// TwinCAT 3 PLC project L2SIVacuum
// Title: LCLS Vacuum
// Company: SLAC - LCLS
// Author: LCLS ECS-Platforms
// ProjectVersion: 0.0.0.0.0.0.
// ProgramVersion: 3.1.4026.17
// libraries:
//   LCLS General, * (SLAC)
//   PMPS, * (SLAC - LCLS)
//   Tc2_DataExchange, * (Beckhoff Automation GmbH)
//   Tc2_EtherCAT, * (Beckhoff Automation GmbH)
//   Tc2_ModbusSrv, * (Beckhoff Automation GmbH)
//   Tc2_SerialCom, * (Beckhoff Automation GmbH)
//   Tc2_Standard, * (Beckhoff Automation GmbH)
//   Tc2_System, * (Beckhoff Automation GmbH)
//   Tc2_TcpIp, * (Beckhoff Automation GmbH)
//   Tc2_Utilities, * (Beckhoff Automation GmbH)
//   Tc3_EventLogger, * (Beckhoff Automation GmbH)
//   Tc3_JsonXml, * (Beckhoff Automation GmbH)
//   Tc3_Module, * (Beckhoff Automation GmbH)
//   TcUnit, * (www.tcunit.org)
// project tree:
//   DUTs/Gauges/ E_PressureState.TcDUT (not stored), Gauge_Type.TcDUT (not stored), ST_VG.TcDUT (not stored)
//   DUTs/LVDT/ ST_SerLVC4000.TcDUT (not stored)
//   DUTs/Oerlikon/ ST_TD20Status.TcDUT (not stored), ST_TD400Control.TcDUT (not stored), ST_TD400Status.TcDUT (not stored)
//   DUTs/Pfeiffer/ ST_PfeifferControl.TcDUT (not stored), ST_PfeifferStatus.TcDUT (not stored)
//   DUTs/Pumps/ E_PumpState.TcDUT (not stored), ST_AgilentPTM.TcDUT (not stored), ST_EbaraDryPump.TcDUT (not stored), ST_EbaraEVA.TcDUT, ST_EbaraPTM.TcDUT (not stored), ST_KashiyamaDryPump.TcDUT (not stored), ST_LeyboldPTM.TcDUT (not stored), ST_PfeifferPTM.TcDUT (not stored), ST_PIP.TcDUT (not stored), ST_PTM.TcDUT (not stored), ST_RoughPump.TcDUT (not stored)
//   DUTs/Valves/ E_ValvePositionState.TcDUT (not stored), E_VCN.TcDUT (not stored), E_2OO3_MODE.TcDUT (not stored), E_VGC.TcDUT (not stored), ST_ValveBase.TcDUT (not stored), ST_VFS.TcDUT (not stored), ST_VGC_2S.TcDUT (not stored), ST_VRC_NO.TcDUT (not stored), ST_VWC_NO.TcDUT (not stored), ST_VVC.TcDUT (not stored), ST_VCC_NO.TcDUT (not stored), ST_VCN.TcDUT (not stored), ST_VGC.TcDUT (not stored), ST_VRC.TcDUT (not stored)
//   DUTs/Valves/VAT590/EtherCAT Interface/ E_ControlMode.TcDUT (not stored), E_ControlModeSP.TcDUT (not stored), E_FatalErrors.TcDUT (not stored), ST_ExtendedWarnings.TcDUT (not stored), ST_GeneralControlSP.TcDUT (not stored), ST_GeneralStatus.TcDUT (not stored), ST_GeneralWarnings.TcDUT (not stored)
//   DUTs/Valves/VAT590/ E_VAT590_AccessMode.TcDUT (not stored), E_VAT590_PID_CTRL.TcDUT (not stored), E_VCN_VAT590.TcDUT (not stored), ST_CoEIndSub.TcDUT (not stored), ST_VAT590_COE.TcDUT, ST_VAT590_STATUS.TcDUT (not stored), ST_VCN_VAT590.TcDUT
//   GVLs/ Constants.TcGVL (not stored), Global_Variables.TcGVL (not stored), GVL_MacroSensorsParameters.TcGVL (not stored), GVL_PfeifferParameters.TcGVL (not stored)
//   / PlcTask.TcTTO (not stored)
//   POUs/ADS/ FB_ADS.TcPOU (not stored), FB_ADS_WATCHDOG.TcPOU (not stored), FB_TBOOL_ADS.TcPOU (not stored)
//   POUs/Functions/Deprecated/Gauges/ FB_MKS317A.TcPOU (not stored), FB_MKS500_EP.TcPOU (not stored), FB_PressureState.TcPOU (not stored)
//   POUs/Functions/Deprecated/Valves/ FB_VCC.TcPOU (not stored), FB_VCC_NO.TcPOU (not stored), FB_VGC_AP.TcPOU (not stored), FB_VGC_EBD.TcPOU (not stored)
//   POUs/Functions/Gauges/ FB_901_ECAT.TcPOU (not stored), FB_9XX.TcPOU (not stored), FB_972.TcPOU (not stored), FB_IE514.TcPOU (not stored), FB_MX7M.TcPOU (not stored), FB_MKS355.TcPOU (not stored), FB_GaugeBase.TcPOU (not stored), FB_CVM201.TcPOU (not stored), FB_CCM501.TcPOU (not stored), FB_IMG401.TcPOU (not stored), FB_MKS909.TcPOU (not stored), FB_MKS909_RBK.TcPOU (not stored), FB_CMR362.TcPOU (not stored), FB_GCM.TcPOU (not stored), FB_ITR90.TcPOU (not stored), FB_MKS392.TcPOU (not stored), FB_MKS500.TcPOU (not stored), FB_MKS722.TcPOU (not stored), FB_MKS_937A.TcPOU (not stored), FB_MKS317.TcPOU (not stored), FB_MKS275.TcPOU (not stored), FB_MKS_937B.TcPOU (not stored), FB_MKS422.TcPOU (not stored)
//   POUs/Functions/Gauges/Interfaces/ FB_GaugeModbus.TcPOU (not stored), FB_Gauge_Interface.TcPOU (not stored), FB_TGCC_ADS.TcPOU (not stored), FB_TGPI_ADS.TcPOU (not stored), FB_GaugeSelection.TcPOU (not stored)
//   POUs/Functions/Pumps/ FB_EbaraDryPump.TcPOU (not stored), FB_EbaraEVA.TcPOU, FB_KashiyamaPump.TcPOU (not stored), FB_KashiyamaPump_G.TcPOU (not stored), FB_PIP_Gamma.TcPOU (not stored), FB_PIP_Gamma_V2.TcPOU, FB_PIP_SIP.TcPOU (not stored), FB_PTM_Agilent.TcPOU (not stored), FB_PTM_Ebara_011M.TcPOU (not stored), FB_PTM_Ebara_010M.TcPOU (not stored), FB_PTM_MagDriveDigital.TcPOU (not stored), FB_PTM_Pfeiffer.TcPOU, FB_PTM_TurboDrive.TcPOU, FB_PTM_TwisTorr.TcPOU (not stored), FB_Pump.TcPOU (not stored), FB_ScrollPump.TcPOU (not stored)
//   POUs/Functions/Pumps/functions/ FB_TurboExtLogic.TcPOU (not stored), F_TurboExtILK_NO.TcPOU (not stored), F_TurboExtILKLogic.TcPOU (not stored), F_TurboExtILKLogic_2.TcPOU (not stored), F_TurboExtILK_NO_1.TcPOU (not stored)
//   POUs/Functions/Pumps/Interfaces/ FB_PIP_Interface_In.TcPOU (not stored), FB_PIP_Interface_Out.TcPOU (not stored), FB_TPIP_ADS.TcPOU (not stored)
//   POUs/Functions/Valves/ FB_Kashiyama_VRC.TcPOU (not stored), FB_MKS248.TcPOU (not stored), FB_TurbVentvalve_NO.TcPOU (not stored), FB_Valve.TcPOU (not stored), FB_VCN_VAT590.TcPOU, FB_VFS.TcPOU (not stored), FB_VFS_2OO3.TcPOU, FB_VGC_NEW.TcPOU, FB_VGC_2S.TcPOU (not stored), FB_VRC_DA.TcPOU (not stored), FB_VRC_EBD.TcPOU (not stored), FB_VRC_NC_ClsLS.TcPOU (not stored), FB_VRC_NO.TcPOU (not stored), FB_VRC_NO_FFO.TcPOU (not stored), FB_VVC.TcPOU (not stored), FB_VCN.TcPOU (not stored), FB_VGC.TcPOU (not stored), FB_VRC.TcPOU (not stored), FB_VRC_OK_CLS.TcPOU (not stored)
//   POUs/Functions/Valves/functions/ F_RoughPumpInlet_ILK.TcPOU (not stored), F_TurboGateValve_ILK.TcPOU (not stored), F_TurboGateValve_ILK_1.TcPOU (not stored), F_TurboGateValve_Protection_ILK.TcPOU (not stored), F_TURBO_VRC_ILK.TcPOU (not stored), F_VALVE_REL_ILK.TcPOU (not stored), F_VRC_DIODE_ILK_OK.TcPOU (not stored), F_VRC_DIODE_ILK.TcPOU (not stored)
//   POUs/Functions/Valves/Interfaces/ FB_TVGC_2S_ADS.TcPOU (not stored), FB_VFS_2OO3Interface.TcPOU, FB_VFS_Interface.TcPOU, FB_TVGC_ADS.TcPOU (not stored), FB_Valve_Interface.TcPOU (not stored), ITF_Valve.TcIO (not stored)
//   POUs/Serial drivers/LVDT/MacroSensors/ FB_LVC4000Com.TcPOU (not stored), FB_LVC4000SerialDriver.TcPOU (not stored), FB_LVC4000Transaction.TcPOU (not stored)
//   POUs/Serial drivers/Pumps/Oerlikon TD20/ FB_OERLIKON_TD20_COM.TcPOU (not stored), FB_OERLIKON_TO_PTM.TcPOU (not stored), FB_TD20SerialDriver.TcPOU (not stored), FB_TD20Transaction.TcPOU (not stored), F_CalcTD20Checksum.TcPOU (not stored)
//   POUs/Serial drivers/Pumps/Oerlikon TD400/ FB_OERLIKON_TD400_COM.TcPOU (not stored), FB_OERLIKON_TD400_TO_PTM.TcPOU (not stored), FB_TD400SerialDriver.TcPOU (not stored), FB_TD400Transaction.TcPOU (not stored), F_CalcTD400Checksum.TcPOU (not stored)
//   POUs/Serial drivers/Pumps/Pfeiffer/ FB_PfeifferSerialDriver.TcPOU (not stored), FB_PfeifferTransaction.TcPOU (not stored), FB_PFEIFFER_COM.TcPOU (not stored), FB_PFEIFFER_TO_PTM.TcPOU (not stored), F_CalcPfeifferCheckSum.TcPOU (not stored)
//   UnitTests/Functions/ V_TO_INT.TcPOU (not stored)
//   UnitTests/Gauges/ FB_GCC_Test.TcPOU (not stored), FB_GHC_Test.TcPOU (not stored), FB_GPI_Test.TcPOU (not stored)
//   UnitTests/ PRG_Test.TcPOU (not stored)
//   UnitTests/Pumps/ FB_PIP_Test.TcPOU (not stored), FB_PTM_Test.TcPOU (not stored)
//   UnitTests/Valves/ FB_VGC_Test.TcPOU (not stored), FB_VRC_Test.TcPOU (not stored)
//   Version/ Global_Version.TcGVL
// real-time tasks:
//   TASK TestTask: cycle T#10ms, priority 16, ADS port 350
// variable links:
//   L2SIVacuum/L2SIVacuum Instance <-> L2SIVacuum/L2SIVacuum Instance
//     PlcTask Inputs/PRG_Test.fb_GCC_Test.fb_MKS422.i_iPRESS_R <-> PlcTask Outputs/PRG_Test.fb_GCC_Test.i_iPRESS_R
//     PlcTask Inputs/PRG_Test.fb_GPI_Test.fb_MKS275.i_iPRESS_R <-> PlcTask Outputs/PRG_Test.fb_GPI_Test.i_iPRESS_R
//     PlcTask Inputs/PRG_Test.fb_GPI_Test.fb_MKS317.i_iPRESS_R <-> PlcTask Outputs/PRG_Test.fb_GPI_Test.i_iPRESS_R
//     PlcTask Inputs/PRG_Test.fb_PTM_Test.fb_PTM_Ebara_010M.i_iCurrentMon <-> PlcTask Outputs/PRG_Test.fb_PTM_Test.i_iCurrentMon
//     PlcTask Inputs/PRG_Test.fb_PTM_Test.fb_PTM_Ebara_010M.i_iRawSpeed <-> PlcTask Outputs/PRG_Test.fb_PTM_Test.i_iRawSpeed
//     PlcTask Inputs/PRG_Test.fb_PTM_Test.fb_PTM_Ebara_010M.i_iTempMon <-> PlcTask Outputs/PRG_Test.fb_PTM_Test.i_iTempMon
//     PlcTask Inputs/PRG_Test.fb_PTM_Test.q_iSpeedSet <-> PlcTask Outputs/PRG_Test.fb_PTM_Test.i_diCurSpd

// ---- DUTs/Pumps/ST_EbaraEVA.TcDUT
TYPE ST_EbaraEVA EXTENDS ST_RoughPump:
STRUCT

(* Output *)
    //q_xRunDO 	:	BOOL; in Rough PUMP


(* Input *)
{attribute 'pytmc' := '
    pv: REMOTE;
    field: ZNAM FALSE;
    field: ONAM TRUE;
    io: io;
    '}
    q_xRemote	:	BOOL;
    {attribute 'pytmc' := '
    pv: ALARM_OK;
    field: ZNAM FALSE;
    field: ONAM TRUE;
    io: i
    '}
    i_xAlarmOK	:	BOOL;

    {attribute 'pytmc' := '
    pv: RUN_DI;
    field: ZNAM FALSE;
    field: ONAM TRUE;
    io: i
    '}
    i_xIsRun		:	BOOL;



END_STRUCT
END_TYPE

// ---- DUTs/Valves/VAT590/ST_VAT590_COE.TcDUT
TYPE ST_VAT590_COE :
STRUCT
    {attribute 'pytmc' := '
    pv: PID_CTRL
    io: io
    '}
    ePIDCtrl: E_VAT590_PID_CTRL;
    (*Adaptive Downstream Parameters*)
    {attribute 'pytmc' := '
    pv: SENS_DELAY_AD
    io: io
    field: EGU "s"
    field: DRVL 0.0
    field: DRVH 1.0
    '}
    fSensorDelay_AD : REAL;
    {attribute 'pytmc' := '
    pv: RAMP_TIME_AD
    io: io
    field: EGU "s"
    field: DRVL 0.0
    field: DRVH 1000000.0
    '}
    fRampTime_AD : REAL;
    {attribute 'pytmc' := '
    pv: RAMP_MODE_AD
    io: io
    field: ZNAM CONST_TIME
    field: ONAM CONST_SLOPE
    '}
    bRampMode_AD : BOOL;
    {attribute 'pytmc' := '
    pv: GAIN_FACTOR_AD
    io: io
    field: PREC 4
    field: DRVL 0.0001
    field: DRVH 7.5
    '}
    fGainFactor_AD : REAL;
    (*Fixed 1 Parameters*)
    {attribute 'pytmc' := '
    pv: RAMP_TIME_FIX1
    io: io
    field: EGU "s"
    field: DRVL 0.0
    field: DRVH 1000000.0
    '}
    fRampTime_FIX1 : REAL;
    {attribute 'pytmc' := '
    pv: RAMP_MODE_FIX1
    io: io
    field: ZNAM CONST_TIME
    field: ONAM CONST_SLOPE
    '}
    bRampMode_FIX1 : BOOL;
    {attribute 'pytmc' := '
    pv: CTRL_DIR_FIX1
    io: io
    field: ZNAM DOWNSTREAM
    field: ONAM UPSTREAM
    '}
    bCtrlDir_FIX1 : BOOL;
    {attribute 'pytmc' := '
    pv: PGAIN_FIX1
    io: io
    field: DRVL 0.001
    field: DRVH 100.0
    '}
    fPGain_FIX1 : REAL;
    {attribute 'pytmc' := '
    pv: IGAIN_FIX1
    io: io
    field: DRVL 0.0
    field: DRVH 100.0
    '}
    fIGain_FIX1 : REAL;
    (*Fixed 2 Parameters*)
    {attribute 'pytmc' := '
    pv: RAMP_TIME_FIX2
    io: io
    field: EGU "s"
    field: DRVL 0.0
    field: DRVH 1000000.0
    '}
    fRampTime_FIX2 : REAL;
    {attribute 'pytmc' := '
    pv: RAMP_MODE_FIX2
    io: io
    field: ZNAM CONST_TIME
    field: ONAM CONST_SLOPE
    '}
    bRampMode_FIX2 : BOOL;
    {attribute 'pytmc' := '
    pv: CTRL_DIR_FIX2
    io: io
    field: ZNAM DOWNSTREAM
    field: ONAM UPSTREAM
    '}
    bCtrlDir_FIX2 : BOOL;
    {attribute 'pytmc' := '
    pv: PGAIN_FIX2
    io: io
    field: DRVL 0.001
    field: DRVH 100.0
    '}
    fPGain_FIX2 : REAL;
    {attribute 'pytmc' := '
    pv: IGAIN_FIX2
    io: io
    field: DRVL 0.0
    field: DRVH 100.0
    '}
    fIGain_FIX2 : REAL;
    (*Soft Pump Parameters*)
    {attribute 'pytmc' := '
    pv: RAMP_TIME_SP
    io: io
    field: EGU "s"
    field: DRVL 0.0
    field: DRVH 1000000.0
    '}
    fRampTime_SP : REAL;
    {attribute 'pytmc' := '
    pv: RAMP_MODE_SP
    io: io
    field: ZNAM CONST_TIME
    field: ONAM CONST_SLOPE
    '}
    bRampMode_SP : BOOL;
    {attribute 'pytmc' := '
    pv: PGAIN_SP
    io: io
    field: DRVL 0.001
    field: DRVH 100.0
    '}
    fPGain_SP : REAL;
END_STRUCT
END_TYPE

// ---- DUTs/Valves/VAT590/ST_VCN_VAT590.TcDUT
TYPE ST_VCN_VAT590 :
STRUCT
    (* VCN - Valve Controlled Needle
    Used for VAT590 needle valves *)
    {attribute 'pytmc' := '
    pv: POS_RAW
    io: i
    '}
    nRawPosition : DINT; //Position readback
    {attribute 'pytmc' := '
    pv: PRES_RAW
    io: i
    '}
    nRawPressure : DINT; //Pressure readback
    {attribute 'pytmc' := '
    pv: PRES_TORR
    field: EGU "TORR"
    io: i
    '}
    fPressure : REAL; //Pressure readback in Torr units
    {attribute 'pytmc' := '
    pv: POS_SP
    io: i
    '}
    nPositionSP : DINT; //Position setpoint readback
    {attribute 'pytmc' := '
    pv: PRES_SP
    io: i
    '}
    nPressureSP : DINT; //Pressure setpoint readback
    {attribute 'pytmc' := '
    pv: ILK_OK
    field: ZNAM NOT OK
    field: ONAM OK
    field: ZSV MAJOR
    field: OSV NO_ALARM
    io: i
    '}
    bIlkOK : BOOL := FALSE; //Interlock Bit status
    {attribute 'pytmc' := '
    pv: POS_LIMIT
    io: io
    autosave_pass1: VAL DESC
    '}
    fPosSetLimit	: REAL := 100; //Percentage Upper limit on valve open
    {attribute 'pytmc' := '
    pv: PRES_SET_LIMIT
    io: io
    autosave_pass1: VAL DESC
    '}
    fPresSetLimit	: REAL := 1E-2; //Upper limit for pressure control
    {attribute 'pytmc' := '
    pv: PRES_RDBK_LIMIT
    io: io
    autosave_pass1: VAL DESC
    '}
    fPresRdbkLimit : REAL := 1E-4;  //Upper limit for pressure reading before valve close
    {attribute 'pytmc' := '
    pv: POS_REQ
    field: DRVL 0.0
    field: DRVH 100.0
    io: io
    '}
    fReqPosition : REAL; //Requested position (0.0-100.0%)
    {attribute 'pytmc' := '
    pv: PRES_REQ
    field: EGU "TORR"
    io: io;
    '}
    fReqPressure : REAL; //Requested pressure in Torr units
    {attribute 'pytmc' :=  '
    pv: STATE
    io: io
    '}
    eValveControl : E_VCN_VAT590; //Valve control mode
    {attribute 'pytmc' := '
    pv:
    '}
    stValveStatus : ST_VAT590_STATUS; //All Valve status readbacks
    {attribute 'pytmc' :=  '
    pv: PRES_SENS
    io: io
    '}
    ePressureSensor : E_VAT590_PressureSensor; //Select pressure sensor
    {attribute 'pytmc' :=  '
    pv: REM_CTRL
    io: io
    '}
    eRemoteControl : E_VAT590_AccessMode; //Select remote control mode
    {attribute 'pytmc' := '
    pv: ZERO
    io: io
    '}
    bZero : BOOL; //Activate Zero function bit
    {attribute 'pytmc' := '
    pv: COE_PARAM
    '}
    stCoeParameters : ST_VAT590_COE; //Coe Parameters
    {attribute 'pytmc' := '
    pv: COE_ERROR
    field: ZNAM OK
    field: ONAM ERROR
    field: ZSV NO_ALARM
    field: OSV MINOR
    io: i
    '}
    bCoeError : BOOL; //Coe Interface Error
    {attribute 'pytmc' := '
    pv: COE_RESET
    io: io
    '}
    bResetCoeError : BOOL; //Reset Coe Interface Error
    {attribute 'pytmc' := '
    pv: ETHCAT_COMM_STATUS
    field: ZNAM OK
    field: ONAM ERROR
    field: ZSV NO_ALARM
    field: OSV MAJOR
    io: i
    '}
    bValveEthCatStatus : BOOL; //Status of the Ethercat Communication with device
END_STRUCT
END_TYPE

// ---- Version/Global_Version.TcGVL
{attribute 'TcGenerated'}
{attribute 'no-analysis'}
{attribute 'linkalways'}
// This function has been automatically generated from the project information.
VAR_GLOBAL CONSTANT
	{attribute 'const_non_replaced'}
	stLibVersion_LCLS_Vacuum : ST_LibVersion := (iMajor := 0, iMinor := 0, iBuild := 0, iRevision := 1, nFlags := 0, sVersion := '0.0.0.1');
END_VAR

// ---- POUs/Functions/Pumps/FB_EbaraEVA.TcPOU
(*This function block does basic controls for the Ebara EV-A  pump. Turns off pump
in the event of errors/ warnings. Provides interlocking interface.*)
FUNCTION_BLOCK FB_EbaraEVA EXTENDS FB_Pump
VAR_INPUT
    i_xExtIlkOK	:	BOOL;
END_VAR
VAR_OUTPUT
    {attribute 'pytmc' := '
    pv:
    '}
    stPump	:	ST_EbaraEVA; //Ebara dry pump structure
END_VAR
VAR
  // For logging
  (*  fbLogger : FB_LogMessage := (eSubsystem:=E_SubSystem.VACUUM);
    ePrevState : E_PumpState;
    tErrorPresent : R_TRIG;
    tAction : R_TRIG; // Primary action of this device (OPN_DO, PUMP_RUN, etc.)
    tFault : F_TRIG;*)

(*IO*)
    q_xRunDo AT%Q* : BOOL; // Output signal
    q_xRemote At%Q* :BOOL;// Remote/Local Control
    q_xResetAlarm At%Q* :BOOL;// Remote/Local Control
    i_xAlarmOK AT%I* :BOOL; // Normally closed Alarm bit
    i_xIsRun   AT%I*:BOOL; // Input status
END_VAR

(*MG 2019*)
stPump.xIlkOK := i_xExtIlkOK AND stPump.i_xAlarmOK ;
// Enable the remote signal when the interlock evaluation is ok
//stPump.q_xRemote := stPump.xIlkOK;

IF stPump.xIlkOK THEN
    stPump.q_xRunDO := stPump.pv_xRunSW;
    stPump.q_xRemote := stPump.pv_xRunSW;
ELSE
        stPump.PV_xRunSW := FALSE;
        stPump.q_xRunDO := FALSE;
END_IF

(*State evaluation*)
IF NOT(stPump.i_xAlarmOK ) THEN
     ePrevState := stpump.eState;
    stpump.eState := pumpFAULT;
ELSIF NOT stpump.q_xRunDo AND stPump.i_xAlarmOK THEN
        stpump.eState := pumpSTOPPED;
ELSIF NOT stpump.q_xRunDo AND NOT stPump.i_xIsRun THEN
        stpump.eState := pumpSTARTING;
ELSIF stPump.i_xIsRun THEN
        stpump.eState := pumpRUNNING;
ELSE
    stpump.eState := pumpFAULT;
END_IF


//Soft IO Mapping
ACT_IO();

// Log States and triggers
ACT_Logger();

ACTION ACT_IO:
stPump.i_xAlarmOK:=	i_xAlarmOK;
stPump.xErr:=	NOT(i_xAlarmOK);
stPump.i_xIsRun := i_xIsRun;
(*outputs*)
q_xRunDo:=stPump.q_xRunDo;
q_xRemote:= stPump.q_xRemote;
END_ACTION

ACTION ACT_Logger:
// ILK logger
IF NOT i_xExtIlkOK AND ePrevState = pumpRUNNING THEN
         fbLogger(sMsg:='Lost external interlock while pump was running.', eSevr:=TcEventSeverity.Critical);
END_IF

//STATE Logger
IF ePrevState <> stpump.eState THEN
      CASE stpump.eState OF
        pumpFAULT:
            fbLogger(sMsg:='Pump Fault.', eSevr:=TcEventSeverity.Critical);
          pumpSTOPPED:
            fbLogger(sMsg:='Pump stopped.', eSevr:=TcEventSeverity.Critical);
        pumpSTARTING:
            fbLogger(sMsg:='Pump starting.', eSevr:=TcEventSeverity.Info);
        pumpRUNNING:
            fbLogger(sMsg:='Pump running.', eSevr:=TcEventSeverity.Info);
      END_CASE
      ePrevState := stpump.eState;
  END_IF

// Log Action
tAction(CLK:=  stPump.q_xRunDo);
IF tAction.Q THEN fbLogger(sMsg:='Pump commanded to start', eSevr:=TcEventSeverity.Info); END_IF


// Log FAULT
tFault(CLK:= stPump.i_xAlarmOK);
IF tFault.Q THEN fbLogger(sMsg:='Pump Lost Alarm OK bit', eSevr:=TcEventSeverity.Critical); END_IF
END_ACTION

END_FUNCTION_BLOCK

// ---- POUs/Functions/Pumps/FB_PIP_Gamma_V2.TcPOU
(* This function block does basic controls FOR the ION pump connected to a Gamma QPCe controller. *)
{attribute 'reflection'}
FUNCTION_BLOCK FB_PIP_Gamma_V2 Extends FB_Pump
VAR_INPUT
END_VAR
VAR_OUTPUT
    {attribute 'pytmc' := '
    pv:
    '}
    stPump	:	ST_PIP; //Gamma Ion pump structure
    q_IG	:	ST_VG; //When ion pump is used as a measuring device for interlocking gate valves
END_VAR
VAR
    rPRESS : REAL;

    rV : REAL;

    (* IO Controls *)
    i_iPRESS  AT %I*: INT;  //
    i_xSP_DI  AT %I* : BOOL; // NO contact //function of relay set on the QPC to HV output state

    // For logging
    tPumpErrorTimeout : TON := (PT:=T#10S); // Timeout pump start if pressure < 1E-11 for more than 10s.

    {attribute 'instance-path'}
    {attribute 'noinit'}
    sPath: STRING;
    fbGetCurTaskIdx  : GETCURTASKINDEX;
    fbWritePersistentData           : WritePersistentData;

END_VAR
VAR CONSTANT
    rMaxPressure : REAL :=1E-4; // Default protection setpoint as per the gamma QPCe manual
    rMinPressure : REAL :=1E-11;
END_VAR
VAR PERSISTENT
END_VAR

(*Pump STATE*)
tPumpErrorTimeout(IN:=(q_IG.rPRESS <= rMinPressure AND stPump.i_xHV_DI));

IF q_IG.rPRESS <= rMinPressure AND stPump.i_xHV_DI THEN
    IF tPumpErrorTimeout.Q THEN
        stPump.eState := pumpFAULT;
        tPumpErrorTimeout(IN:=FALSE);
    END_IF
ELSIF q_IG.rPRESS <= rMinPressure AND NOT stPump.i_xHV_DI THEN
    stPump.eState := pumpSTOPPED;
ELSIF stPump.i_xHV_DI THEN
    stPump.eState := pumpRUNNING;
ELSE
    stPump.eState := pumpFAULT;
END_IF

(*Update output gauge values*)
ACT_SetGauge();
(*Soft IO Mapping*)
IO();
// Log States and triggers
ACT_Logger();

ACTION ACT_Logger:
//STATE Logger
IF ePrevState <> stPump.eState THEN
      CASE stPump.eState OF
        pumpFAULT:
            fbLogger(sMsg:='Pump Fault.', eSevr:=TcEventSeverity.Critical);
        pumpSTOPPED:
            fbLogger(sMsg:='Pump stopped.', eSevr:=TcEventSeverity.Critical);
        pumpRUNNING:
            fbLogger(sMsg:='Pump running.', eSevr:=TcEventSeverity.Info);
      END_CASE
      ePrevState := stPump.eState;
  END_IF
END_ACTION

ACTION ACT_SetGauge:
(*MG*)
(* convert the analog input into readable pressure*)
(* use logarithmic Pressure calculation, Output= Normal and Offset = 0*)
rV := 10*INT_TO_REAL(i_iPress)/32767;
//Manual Page 9

if (stPump.bOutputInverted) THEN
    rPRESS := LREAL_TO_REAL(EXPT(10,(rV-stPump.iOffset)*-1));
ELSE
    rPRESS := LREAL_TO_REAL(EXPT(10,(rV-stPump.iOffset)));
END_IF

q_IG.rPRESS := rPRESS;
stPump.rPRESS := rPRESS;

IF stPump.eState := pumpRUNNING THEN
    q_IG.xPRESS_OK := TRUE;
ELSE
    q_IG.xPRESS_OK := FALSE;
END_IF

q_IG.sPath := This^.stPump.sPath;
END_ACTION

ACTION IO:
stPump.xError := (stPump.eState = pumpFAULT);

(*inputs*)
stPump.i_iPRESS:=	i_iPRESS;
stPump.i_xHV_DI:=	i_xSP_DI;

 This^.stPump.sPath:= sPath;
END_ACTION

END_FUNCTION_BLOCK

// ---- POUs/Functions/Pumps/FB_PTM_Pfeiffer.TcPOU
(* This function block does basic controls FOR the Pfeiffer Turbo pump connected to the TM700 and TC400 Controllers.
 Turns off pump in the event of errors/ warnings. Provides interlocking interface.*)
FUNCTION_BLOCK FB_PTM_Pfeiffer EXTENDS FB_Pump
VAR_INPUT
    i_xExtIlkOK : BOOL; // Connect to external interlock logic, TRUE if not used.
END_VAR
VAR_OUTPUT
    {attribute 'pytmc' := '
    pv:
    '}
    iq_stPTM : ST_PfeifferPTM;
END_VAR
VAR
    TOF_RESET: TON :=(PT:=T#1S);
    (*IO*)
    i_xAtSpd AT%I*: BOOL; // Normaml operation when true
    i_xFaultNC AT%I*: BOOL; // Error
    i_xWarn AT%I*: BOOL;
     i_xRemote AT%I*: BOOL;

    q_RunDO AT%Q*: BOOL; // Start/Stop for TC110 link this output to the Pumping station bit
    q_PumpingStation AT%Q*: BOOL; // Start/Stop interlock
    q_xRemote AT%Q*: BOOL;
    q_xReset AT%Q*: BOOL;
END_VAR

(* Basic pump supervisory section *)

q_xRemote := TRUE;
(* Interlock Sum *)
iq_stPtm.xExtRunOk:= i_xExtILKOk;
//For compatability with TC110
(*IF iq_stPTM.xExtRunOk THEN
    q_PumpingStation:= TRUE;
ELSE
    q_PumpingStation:= FALSE;
END_IF*)

IF iq_stPTM.xExtRunOk AND NOT (iq_stPTM.i_xFault) (*OR iq_stPTM.i_xTempFault)*) THEN
    iq_stPTM.q_RunDO:=iq_stPTM.xRunSW;
    q_PumpingStation:=iq_stPTM.xRunSW;
ELSE
    iq_stPTM.xRunSW:=FALSE;
    iq_stPTM.q_RunDO:=FALSE;
    q_PumpingStation:=FALSE;
END_IF


(*Pump STATE*)
IF iq_stPtm.i_xFault THEN
    iq_stPtm.eState := pumpFAULT;
ELSIF NOT iq_stPtm.q_RunDO AND NOT iq_stPTM.i_xFault THEN
    iq_stPtm.eState := pumpSTOPPED;
ELSIF NOT iq_stPtm.i_xAtSpd  AND iq_stPtm.q_RunDO THEN
    iq_stPtm.eState := pumpSTARTING;
ELSIF iq_stPtm.i_xAtSpd AND iq_stPtm.q_RunDO THEN
    iq_stPtm.eState := pumpRUNNING;
ELSE
    iq_stPtm.eState := pumpFAULT;
END_IF

(*Error Reset*)
(* to reset the Reset Bit *)
 IF (iq_stPTM.xResetSW ) THEN
    iq_stPTM.q_xReset := TRUE;
    q_PumpingStation := TRUE;
 END_IF

 IF (iq_stPTM.xResetSW) AND (iq_stPTM.i_xFault)  THEN
    q_PumpingStation := TRUE;
 END_IF
 TOF_RESET (IN:= iq_stPTM.q_xReset, Q => );
 IF TOF_RESET.Q THEN
    iq_stPTM.q_xReset:= FALSE;
    iq_stPTM.xResetSW := FALSE;
 END_IF

(*Soft IO Mapping*)
ACT_IO();
// Log States and triggers
ACT_Logger();
(*Load or save the persistent variables*)
ACT_Persistent();

ACTION ACT_IO:
(*outputs*)
q_RunDO := iq_stPTM.q_RunDO;
q_xReset := iq_stPTM.q_xReset;
//q_xRemote := iq_stPTM.
//q_PumpingStation AT%Q*: BOOL; // Start/Stop

(*inputs*)
iq_stPTM.i_xAtSpd:= i_xAtSpd;
iq_stPTM.i_xFault:= NOT i_xFaultNC;
iq_stPTM.i_xWarn:=  	i_xWarn ;
END_ACTION

ACTION ACT_Logger:
//STATE Logger
IF NOT i_xExtIlkOK AND ePrevState = pumpRUNNING THEN
         fbLogger(sMsg:='Lost external interlock while pump was running.', eSevr:=TcEventSeverity.Critical);
END_IF


IF ePrevState <> iq_stPTM.eState THEN
      CASE iq_stPTM.eState OF
        pumpFAULT:
            fbLogger(sMsg:='Pump Fault.', eSevr:=TcEventSeverity.Critical);
          pumpSTOPPED:
            fbLogger(sMsg:='Pump stopped.', eSevr:=TcEventSeverity.Critical);
        pumpSTARTING:
            fbLogger(sMsg:='Pump starting.', eSevr:=TcEventSeverity.Info);
        pumpRUNNING:
            fbLogger(sMsg:='Pump running.', eSevr:=TcEventSeverity.Info);
      END_CASE
      ePrevState := iq_stPTM.eState;
  END_IF

// ILK logger



// Log Action
tAction(CLK:=  iq_stPTM.q_RunDO);
IF tAction.Q THEN fbLogger(sMsg:='Pump commanded to start', eSevr:=TcEventSeverity.Info); END_IF


// Log FAULT
tFault(CLK:= NOT iq_stPTM.i_xFault);
IF tFault.Q THEN fbLogger(sMsg:='Pump Lost Alarm OK bit', eSevr:=TcEventSeverity.Critical); END_IF
END_ACTION

ACTION ACT_Persistent:
(*On first PLC pass, load the persistent value into the structrue variable*)
IF (SUPER^.bRestorePersistentData) THEN
    SUPER^.bRestorePersistentData	:= FALSE;
    IF (rBackingPressureSP <> 0) THEN
        iq_stPTM.rBackingPressureSP := rBackingPressureSP;
    END_IF;
    IF (rInletPressureSP <> 0) THEN
        iq_stPTM.rInletPressureSP := rInletPressureSP;
    END_IF;
END_IF
(*Check if a new value has been written in the structure variable copy it to the persistent variable*)
IF NOT (iq_stPTM.rBackingPressureSP = rBackingPressureSP) THEN
    rBackingPressureSP:= iq_stPTM.rBackingPressureSP;
END_IF;

IF NOT (iq_stPTM.rInletPressureSP = rInletPressureSP) THEN
    rInletPressureSP := iq_stPTM.rInletPressureSP;
END_IF;
END_ACTION

METHOD PUBLIC M_Run : BOOL
VAR_INPUT
    run:bool; // set to true to run, false to stop;
END_VAR

this^.iq_stPtm.xRunSW := run;
END_METHOD

METHOD PUBLIC M_Serial_IO : BOOL
VAR_INPUT
    st_Pfeiffer_RBK: ST_PfeifferStatus;
END_VAR
VAR_IN_OUT
    st_Pfeiffer_CTRL: ST_PfeifferControl;
END_VAR
(* This function block is used to map the IO points from the pfeiffer structures
to the generic turbo structures *)
(*
if (bInit) Then
    bInit := False;
    st_Pfeiffer_CTRL.diSetRotationSpeed_309 := st_Pfeiffer_RBK.diActiveRotationSpeed_309;
END_IF*)

(* Controls *) (* Controls is via DIO*)
//st_Pfeiffer_CTRL.xPumpingStation_010 := iq_stPTM.q_RunDO;
//st_Pfeiffer_CTRL.xMotorPump_023 := 1; //Setting always true because parameter 10 alone can enable/disable the pump
//st_Pfeiffer_CTRL.uiPowerPct_708 := iq_stPTM.q_uiPowerPct;
//st_Pfeiffer_CTRL.xErrorAck_009 := iq_stPTM.xResetSW;



(* Readbacks *)
iq_stPTM.i_xAccel := st_Pfeiffer_RBK.xPumpAccelerating_307;
//iq_stPTM.i_xAtSpd := st_Pfeiffer_RBK.xRotationSpeedAttn_306; The Atspd is already linked via Digital I/Os
iq_stPTM.i_diCurSpd := st_Pfeiffer_RBK.diActiveRotationSpeed_309;
iq_stPTM.i_diPwr := st_Pfeiffer_RBK.diDrivePower_316;
iq_stPTM.i_diElecTemp := st_Pfeiffer_RBK.diTempElec_326;
iq_stPTM.i_diBtmTemp := st_Pfeiffer_RBK.diTempPmpBot_330;
iq_stPTM.i_diBrngTemp := st_Pfeiffer_RBK.diTempBearng_342;
iq_stPTM.i_diMtrTemp := st_Pfeiffer_RBK.diTempMotor_346;
iq_stPTM.i_uiPowerPctRbk := st_Pfeiffer_RBK.uiPowerPct_708;
iq_stPTM.i_rCurrentMon :=  st_Pfeiffer_RBK.lrDriveCurrent_310;
iq_stPTM.xCommTimeout	:=	st_Pfeiffer_RBK.xTimeout;
iq_stPTM.i_iErrorCode := st_Pfeiffer_RBK.iErrorCode_303;
iq_stPTM.i_iWarningCode := st_Pfeiffer_RBK.iWarningCode_303;

(* Check that error acknowledgment is processed *)
IF st_Pfeiffer_RBK.xErrorAcknowledged THEN
    st_Pfeiffer_RBK.xErrorAcknowledged := FALSE;
    st_Pfeiffer_CTRL.xErrorAck_009 := FALSE;
    iq_stPTM.xResetSW := FALSE;
END_IF

IF st_Pfeiffer_RBK.sErrorCode_303 = '' THEN
    ;
ELSIF st_Pfeiffer_RBK.sErrorCode_303 <> '000000' THEN
iq_stPTM.i_xFault := TRUE;
ELSE
iq_stPTM.i_xFault := FALSE;
END_IF

st_Pfeiffer_CTRL.xSetSpdMode_026:= iq_stPTM.q_bSetSpd;
iq_stPTM.i_dSetSpd := LIMIT (0, iq_stPTM.i_dSetSpd, 1500); // 1500 nominal frequency
IF ( iq_stPTM.i_dSetSpd <>0) THEN
    st_Pfeiffer_CTRL.iSetRotationSpeed_707 := DINT_TO_INT(iq_stPTM.i_dSetSpd * 100/1500);
    st_Pfeiffer_CTRL.iSetRotationSpeed_707 := LIMIT(20, st_Pfeiffer_CTRL.iSetRotationSpeed_707 ,100); // Manual Page 18
END_IF
END_METHOD

END_FUNCTION_BLOCK

// ---- POUs/Functions/Pumps/FB_PTM_TurboDrive.TcPOU
(* This Function block provides basic turbo control for Leybold Turbo Drive 300, Turbo Drive 400 *)
(* TD20 Classic Via Remote X1 Connector 9-way PLC interface*)
(* When serial interface is implemented, call Method M_Serial_IO after fb instantiation, in order to add the serial status *)
FUNCTION_BLOCK FB_PTM_TurboDrive EXTENDS FB_Pump
VAR_INPUT
    i_xExtILKOk : BOOL; // Connect to external interlock logic, TRUE if not used.
END_VAR
VAR_OUTPUT
    {attribute 'pytmc' := '
    pv:
    '}
    iq_stPtm	:	ST_LeyboldPTM;
END_VAR
VAR

    xRunOk	:	BOOL;
    tofRemoteDelay	:	TOF;


    (*IO*)
    i_xAtSpd AT%I*: BOOL; // Normaml operation when true
    i_xFaultNC AT%I*: BOOL; // Error Active when no Error is present
    q_RunDO AT%Q*: BOOL; // Start/Stop
END_VAR

(* Basic Turbo Control *)
(* This Function block provides basic turbo control for Leybold Turbo Drive 300, Turbo Drive 400 *)
(* TD20 Classic Via Remote X1 Connector 9-way PLC interface*)
(* M. Ghaly Jan. 2019 *)

(* Interlock Sum *)
iq_stPtm.xExtRunOk:= i_xExtILKOk;
xRunOk := iq_stPtm.xExtRunOk AND iq_stPtm.i_xNCError;

(* Basic pump supervisory section *)
IF xRunOk THEN
    q_RunDO := iq_stPTM.xRunSW;
ELSE
    iq_stPtm.xRunSW:=FALSE;
    q_RunDO:=FALSE;
END_IF

(*Pump States*)
IF (iq_stPtm.i_xFault) THEN
        iq_stPtm.eState := pumpFAULT;
        iq_stPtm.xRunSW:=FALSE;
        q_RunDO:=FALSE;
ELSIF (iq_stPtm.q_RunDO) AND (iq_stPtm.i_xAtSpd) THEN
        iq_stPtm.eState := pumpRUNNING;
ELSIF (iq_stPtm.q_RunDO) AND NOT (iq_stPtm.i_xAtSpd) THEN
        iq_stPtm.eState := pumpSTARTING;
ELSIF NOT (iq_stPtm.q_RunDO) THEN
        iq_stPtm.eState := pumpSTOPPED;
ELSE
    iq_stPtm.eState := pumpFAULT;
END_IF;


(*I/O soft mapping*)
ACT_IO();
// Log States and triggers
This^.ACT_Logger();
(*Load or save the persistent variables*)
ACT_Persistent();

ACTION ACT_IO:
(*Inputs*)
iq_stPtm.i_xAtSpd := i_xAtSpd;
iq_stPtm.i_xNCError := i_xFaultNC;
iq_stPtm.i_xFault := NOT i_xFaultNC;



(*Outputs*)
iq_stPtm.q_RunDO := q_RunDO;
END_ACTION

ACTION ACT_Logger:
//STATE Logger
// ILK logger
IF NOT i_xExtIlkOK AND ePrevState = pumpRUNNING THEN
         fbLogger(sMsg:='Lost external interlock while pump was running.', eSevr:=TcEventSeverity.Critical);
END_IF


IF ePrevState <> iq_stPTM.eState THEN
      CASE iq_stPTM.eState OF
        pumpFAULT:
            fbLogger(sMsg:='Pump Fault.', eSevr:=TcEventSeverity.Critical);
          pumpSTOPPED:
            fbLogger(sMsg:='Pump stopped.', eSevr:=TcEventSeverity.Critical);
        pumpSTARTING:
            fbLogger(sMsg:='Pump starting.', eSevr:=TcEventSeverity.Info);
        pumpRUNNING:
            fbLogger(sMsg:='Pump running.', eSevr:=TcEventSeverity.Info);
      END_CASE
      ePrevState := iq_stPTM.eState;
  END_IF

// Log Action
tAction(CLK:=  iq_stPTM.q_RunDO);
IF tAction.Q THEN fbLogger(sMsg:='Pump commanded to start', eSevr:=TcEventSeverity.Info); END_IF


// Log FAULT
tFault(CLK:= NOT iq_stPTM.i_xFault);
IF tFault.Q THEN fbLogger(sMsg:='Pump Lost Alarm OK bit', eSevr:=TcEventSeverity.Critical); END_IF
END_ACTION

ACTION ACT_Persistent:
(*On first PLC pass, load the persistent value into the structrue variable*)
IF (SUPER^.bRestorePersistentData) THEN
    SUPER^.bRestorePersistentData	:= FALSE;
    IF (rBackingPressureSP <> 0) THEN
        iq_stPTM.rBackingPressureSP := rBackingPressureSP;
    END_IF;
    IF (rInletPressureSP <> 0) THEN
        iq_stPTM.rInletPressureSP := rInletPressureSP;
    END_IF;
END_IF
(*Check if a new value has been written in the structure variable copy it to the persistent variable*)
IF NOT (iq_stPTM.rBackingPressureSP = rBackingPressureSP) THEN
    rBackingPressureSP:= iq_stPTM.rBackingPressureSP;
END_IF;

IF NOT (iq_stPTM.rInletPressureSP = rInletPressureSP) THEN
    rInletPressureSP := iq_stPTM.rInletPressureSP;
END_IF;
END_ACTION

METHOD PUBLIC M_Run : BOOL
VAR_INPUT
    run:bool; // set to true to run, false to stop;
END_VAR

this^.iq_stPtm.xRunSW := run;
END_METHOD

METHOD PUBLIC M_Serial_IO : BOOL
VAR_INPUT
    i_st_TD20_RBK			: ST_TD20Status;
END_VAR

(* This function block is used to map the IO points from the Oerlikon structures
to the generic turbo structures *)

(* Readbacks *)
iq_stPTM.i_xAccel := i_st_TD20_RBK.wStatusWord.4;
iq_stPTM.i_xDecel := i_st_TD20_RBK.wStatusWord.5;
//iq_stPTM.i_xAtSpd := i_st_TD20_RBK.wStatusWord.10;
iq_stPTM.i_xRemote := i_st_TD20_RBK.wStatusWord.15; (* Remote control enabled *)
iq_stPTM.i_diCurSpd := WORD_TO_DINT(i_st_TD20_RBK.wFrequency_P3);
iq_stPTM.i_rCurrentMon := WORD_TO_INT(i_st_TD20_RBK.wMotorCurrent_P5);
iq_stPTM.i_diPwr := WORD_TO_DINT(i_st_TD20_RBK.wMotorCurrent_P5 * i_st_TD20_RBK.wVoltage_P4);
iq_stPTM.i_diElecTemp := WORD_TO_DINT(i_st_TD20_RBK.wConverterTemp_P11);
iq_stPTM.i_rTempMon := WORD_TO_INT(i_st_TD20_RBK.wPumpTemp_P127);

(* Faults and warnings *)
//iq_stPTM.i_xFault := i_st_TD20_RBK.wStatusWord.3;
iq_stPTM.i_xTempFault := i_st_TD20_RBK.wStatusWord.7; (* specified as a temperature warning but it could be a fault *)
iq_stPTM.i_xWarn := i_st_TD20_RBK.wStatusWord.14; (* warning summary bit *)
END_METHOD

END_FUNCTION_BLOCK

// ---- POUs/Functions/Valves/FB_VCN_VAT590.TcPOU
(* This function implements the Basic functions for the VAT590 needle valve*)
FUNCTION_BLOCK FB_VCN_VAT590 EXTENDS FB_Valve
VAR_INPUT
    bExtIlkOK : BOOL;        // External Interlock, SET to TRUE if not used
    IG : ST_VG;              // Input from a cold cathode gauge used in control loop
END_VAR
VAR_OUTPUT
    {attribute 'pytmc' := '
    pv:
    '}
    stVcnVat590	: ST_VCN_VAT590;       // Needle valve VAT590 structure
END_VAR
VAR CONSTANT
    cOpenPosition : REAL := 1E+5;      // Default position setpoint upper scale value
    cClosePosition : REAL := 0.0;      // Default position setpoint lower scale value
    cPresSPUpLim : REAL := 1E+6;       // Default pressure setpoint upper scale value
    cPresSPLowLim : REAL := 0;         // Default pressure setpoint lower scale value
    cPressCtrl : ST_CoEIndSub := (nIndex := 16#2199, nSubIndex := 0); // Selected pressure controller CoE register
    cSensorDelay_AD : ST_CoEIndSub := (nIndex := 16#219A, nSubIndex := 0); // Adaptive DS controller Sensor Delay CoE register
    cRampTime_AD : ST_CoEIndSub := (nIndex := 16#219B, nSubIndex := 0); // Adaptive DS controller Ramp Time CoE register
    cRampMode_AD : ST_CoEIndSub := (nIndex := 16#219C, nSubIndex := 0); // Adaptive DS controller Ramp Mode CoE register
    cGainFactor_AD : ST_CoEIndSub := (nIndex := 16#219E, nSubIndex := 0); // Adaptive DS controller Gain factor CoE register
    cRampTime_FIX1 : ST_CoEIndSub := (nIndex := 16#21A5, nSubIndex := 0); // Fixed 1 controller Ramp Time CoE register
    cRampMode_FIX1 : ST_CoEIndSub := (nIndex := 16#21A6, nSubIndex := 0); // Fixed 1 controller Ramp Mode CoE register
    cCtrlDir_FIX1 : ST_CoEIndSub := (nIndex := 16#21A7, nSubIndex := 0); // Fixed 1 controller Control Direction CoE register
    cPGain_FIX1 : ST_CoEIndSub := (nIndex := 16#21A8, nSubIndex := 0); // Fixed 1 controller P Gain CoE register
    cIGain_FIX1 : ST_CoEIndSub := (nIndex := 16#21A9, nSubIndex := 0); // Fixed 1 controller I Gain CoE register
    cRampTime_FIX2 : ST_CoEIndSub := (nIndex := 16#21AF, nSubIndex := 0); // Fixed 2 controller Ramp Time CoE register
    cRampMode_FIX2 : ST_CoEIndSub := (nIndex := 16#21B0, nSubIndex := 0); // Fixed 2 controller Ramp Mode CoE register
    cCtrlDir_FIX2 : ST_CoEIndSub := (nIndex := 16#21B1, nSubIndex := 0); // Fixed 2 controller Control Direction CoE register
    cPGain_FIX2 : ST_CoEIndSub := (nIndex := 16#21B2, nSubIndex := 0); // Fixed 2 controller P Gain CoE register
    cIGain_FIX2 : ST_CoEIndSub := (nIndex := 16#21B3, nSubIndex := 0); // Fixed 2 controller I Gain CoE register
    cRampTime_SP : ST_CoEIndSub := (nIndex := 16#21B9, nSubIndex := 0); // Soft Pump controller Ramp Time CoE register
    cRampMode_SP : ST_CoEIndSub := (nIndex := 16#21BA, nSubIndex := 0); // Soft Pump controller Ramp Time CoE register
    cPGain_SP : ST_CoEIndSub := (nIndex := 16#21BC, nSubIndex := 0); // Soft Pump controller Ramp Time CoE register
END_VAR
VAR
    fCalcPosSP : REAL := 0;
    fCalcPresSP : REAL := 0;
    eValveModeSP : E_ControlModeSP;
    fReqPos : REAL;                    // Requested position internal variable
    fReqPres : REAL;                   // Requested pressure internal variable
    fPresLowLim : REAL := 1E-10;       // Pressure sensor lower scale value
    fSlope : REAL := 1E+5;             // Slope (Units per decade) used for conversion from Torr units
    fVbase : REAL := 1E+5;             // Vbase (Units per decade) defined for how much the curve is shifted
    bRemAcsToggle : BOOL;              // Remote access control bit
    //timer for zero function
    tZeroTogg : TON := (PT := T#1S);
    //timer for remote function
    tRemAcsTogg : TON := (PT := T#500MS);
    //used for logging
    ePreviousState : E_VCN_VAT590;

    (*CoE Interface*)
    (*Link this to your VAT590 reference variables under InfoData.*)
    //Connect i_stVat590PlcDriveRef.aNetId to the VAT590 Valve InfoData^AdsAddr^netId
    //Connect i_stVat590PlcDriveRef.nSlaveAddr to the VAT590 Valve InfoData^AdsAddr^port
    i_stVat590PlcDriveRef AT %I*: ST_PlcDriveRef;
    stVat590DriveRef : ST_DriveRef;

    fbCoeRead : FB_CoERead_ByDriveRef;   // CoE Read function block
    fbCoeWrite : FB_CoEWrite_ByDriveRef; // CoE Write function block

    stCoeParamsInternal : ST_VAT590_COE;   // Internal storage of CoE parameters
    nCaseReadCoe : UINT := 1;          // Iterator for going through all CoE parameters
    rtCoeReset : R_TRIG;               // Rising edge trigger for reset CoE Interface error
    ftCoeReadBusy : F_TRIG;            // Falling edge trigger for CoE read new data
    ftCoeWriteBusy : F_TRIG;           // Falling edge trigger for CoE write data
    bFirstRead : BOOL := TRUE;         // FALSE after succesfull first readout of all CoE parameters

    (*VAT590 Ethercat IO Interface*)
    // Ethercat Interface Inputs
    i_nRawPosition       AT %I* : DINT;               // Position readback from the valve
    i_nRawPressure       AT %I* : DINT;               // Pressure readback from the valve
    i_eControlMode       AT %I* : E_ControlMode;      // Valve control mode readback
    i_eFatalError        AT %I* : E_FatalErrors;      // Valve Fatal Errors readback
    i_stGenStatus        AT %I* : ST_GeneralStatus;   // Valve General Status readback
    i_stGenWarnings      AT %I* : ST_GeneralWarnings; // Valve General Warnings readback
    i_stExtnWarnings     AT %I* : ST_ExtendedWarnings;// Valve Extended Warnings readback
    // Ethercat Interface Outputs
    o_nRawPositionSP     AT %Q* : DINT;               // Position setpoint
    o_nRawPressureSP     AT %Q* : DINT;               // Pressure setpoint
    o_eCtrlModeSP        AT %Q* : E_ControlModeSP;    // Valve control mode setpoint
    o_stGenCtrlSP        AT %Q* : ST_GeneralControlSP;// General Control setpoint
    (*Ethercat Interface Status Check*)
    (*Link this to your VAT590 WcState variable under WcState*)
    i_bValveEthCatStatus AT %I* : BOOL := TRUE;
END_VAR
VAR PERSISTENT
    fUpperLimit	: REAL;                // Max position in % that can be requested
    fPresMaxLim : REAL;                // Max pressure in Torr that can be requested
    fPresRbMaxLim : REAL;              // Max pressure in Torr read by chamber gauge, valve will close above the pressure.
END_VAR

(* Needle valve control FB
J. Govednik 2021-11-22

This FB should be used as a low level control block.

It provides:
Valve position ceiling
Interlock
CoE Interface

It could be used for:
Valve position/flow linearization
*)

(*Set Coe Interface, AmsNetID, Slave address etc*)
SetCoeInterface();

(*Read from EPICS and Valve Ethercat interface*)
ReadFromInput();

(*Checking which Control mode is selected and if valve's communication is OK*)
IF stVcnVat590.bValveEthCatStatus THEN //If valve is not connected or something is wrong with EtherCAT communication PLC will set this bit to 1
    fReqPos := 0; //set req. position to 0
    eValveModeSP := E_ControlModeSP.CloseValve; //set control mode of the valve to CLOSE VALVE
    stVcnVat590.eValveControl := E_VCN_VAT590.CloseValve; //EPICS command hold in CloseValve state
    stVcnVat590.stValveStatus.eControlMode := E_ControlMode.FatalError; //override the readback from the valve because when valve is disconnected the value remains
    stVcnVat590.nRawPosition := 0; //override the readback from the valve because when valve is disconnected the value remains
    stVcnVat590.nRawPressure := 0; //override the readback from the valve because when valve is disconnected the value remains
ELSIF bExtIlkOK THEN
    CASE stVcnVat590.eValveControl OF
        E_VCN_VAT590.OpenValve:
            eValveModeSP := E_ControlModeSP.OpenValve;
        E_VCN_VAT590.CloseValve:
            eValveModeSP := E_ControlModeSP.CloseValve;
        E_VCN_VAT590.ManualControl:
            IF IG.xPRESS_OK AND IG.rPRESS <= fPresRbMaxLim THEN
                eValveModeSP := E_ControlModeSP.ManualControl;
            ELSE
                eValveModeSP := E_ControlModeSP.CloseValve; // Close valve if something is wrong with the gauge
                stVcnVat590.eValveControl := E_VCN_VAT590.CloseValve;
            END_IF
        E_VCN_VAT590.PressureControl:
            IF IG.xPRESS_OK AND IG.rPRESS <= fPresRbMaxLim THEN
                eValveModeSP := E_ControlModeSP.PressureControl;
            ELSE
                eValveModeSP := E_ControlModeSP.CloseValve; // Close valve if something is wrong with the gauge
                stVcnVat590.eValveControl := E_VCN_VAT590.CloseValve;
            END_IF
        E_VCN_VAT590.HoldValve:
            IF stVcnVat590.stValveStatus.eControlMode = E_ControlMode.ManualControl OR
                stVcnVat590.stValveStatus.eControlMode = E_ControlMode.PressureControl THEN
                eValveModeSP := E_ControlModeSP.HoldValve;
            END_IF
    END_CASE
ELSE
    fReqPos := 0;
    eValveModeSP := E_ControlModeSP.CloseValve;
    stVcnVat590.eValveControl := E_VCN_VAT590.CloseValve;
END_IF

(*Requested Position calculation*)
fReqPos := LIMIT(0, fReqPos, fUpperLimit);
fCalcPosSP := fReqPos * (cOpenPosition-cClosePosition)/100 + cClosePosition;
fCalcPosSP := LIMIT(cClosePosition, fCalcPosSP, cOpenPosition); //The requested position SP should remain within this range

(*Pressure calculation*)
//Limit the input from EPICS between upper and lower limit defined for seleceted pressure sensor
fReqPres := LIMIT(fPresLowLim, fReqPres, fPresMaxLim);

// Calculate pressure readback and pressure setpoint according to selected pressure gauge
CASE stVcnVat590.ePressureSensor OF
    E_VAT590_PressureSensor.MKS500:
        fPresLowLim := 1.0E-10;
        fSlope := 1E+5;
        fVbase := 1E+5;
        //Calcuate pressure setpoint
        fCalcPresSP := fSlope * LOG(fReqPres/fPresLowLim) + fVbase;
        fCalcPresSP := LIMIT(cPresSPLowLim, fCalcPresSP, cPresSPUpLim); //The requested pressure SP should remain within this range
        //Calculate pressure readback in Torr units
        stVcnVat590.fPressure := LREAL_TO_REAL(EXPT(10,((DINT_TO_REAL(stVcnVat590.nRawPressure)-fVbase)/fSlope + LOG(fPresLowLim))));
    ELSE
        fCalcPresSP := 0;
        stVcnVat590.fPressure := 0;
END_CASE

(*Calculated Pressure SP and Pressure readback is 0 if Pressure sensor is not working*)
IF NOT (IG.xPRESS_OK AND IG.rPRESS < fPresRbMaxLim ) THEN
    fCalcPresSP := 0;
    stVcnVat590.fPressure := 0;
END_IF

(*Zero function*)
IF stVcnVat590.stValveStatus.bZeroDisabled OR tZeroTogg.Q THEN
    stVcnVat590.bZero := FALSE;
END_IF
tZeroTogg.IN := stVcnVat590.bZero;
tZeroTogg();

(*Set Remote Access*)
IF stVcnVat590.stValveStatus.eRemoteStatus <> stVcnVat590.eRemoteControl THEN
    tRemAcsTogg.IN := TRUE;
    IF tRemAcsTogg.Q THEN
        bRemAcsToggle := NOT bRemAcsToggle;
        tRemAcsTogg.IN := FALSE;
    END_IF
END_IF
tRemAcsTogg();

(*Reset Coe Interface error*)
rtCoeReset(CLK := stVcnVat590.bResetCoeError);
IF rtCoeReset.Q THEN
    stVcnVat590.bResetCoeError := FALSE;
END_IF

(*Write CoE Parameters*)
WriteCoeParameters();

(*Read CoE Parameters*)
ReadCoeParameters();

(*Write to EPICS and Valve Ethercat interface*)
WriteToOutput();

(*Load or save the persistent variables*)
LoadPersistentData();

(*Logging*)
Logger();

ACTION LoadPersistentData:
(*On first PLC pass, load the persistent value into the structrue variable*)
IF (bRestorePersistentData) THEN
    bRestorePersistentData	:= FALSE;
    IF (fUpperLimit <> 0) THEN
        stVcnVat590.fPosSetLimit := fUpperLimit;
    END_IF;
    IF (fPresMaxLim <> 0) THEN
        stVcnVat590.fPresSetLimit := fPresMaxLim;
    END_IF;
    IF (fPresRbMaxLim <> 0) THEN
        stVcnVat590.fPresRdbkLimit := fPresRbMaxLim;
    END_IF;
END_IF
END_ACTION

ACTION Logger:
// ILK logger
IF NOT (stVcnVat590.bIlkOK ) AND NOT(ePreviousState = E_VCN_VAT590.CloseValve) THEN
         fbLogger(sMsg:='Lost interlock ok bit while valve was open.', eSevr:=TcEventSeverity.Critical);
END_IF


//Control STATE Logger
IF ePreviousState <> stVcnVat590.eValveControl THEN
      CASE stVcnVat590.eValveControl OF
        E_VCN_VAT590.ManualControl:
            fbLogger(sMsg:='Valve in manual control mode.', eSevr:=TcEventSeverity.Warning);
        E_VCN_VAT590.HoldValve:
            fbLogger(sMsg:='Valve in hold control mode.', eSevr:=TcEventSeverity.Warning);
        E_VCN_VAT590.OpenValve:
            fbLogger(sMsg:='Valve Open.', eSevr:=TcEventSeverity.Info);
        E_VCN_VAT590.PressureControl:
            fbLogger(sMsg:='Valve in pressure control mode.', eSevr:=TcEventSeverity.Info);
        E_VCN_VAT590.CloseValve:
            fbLogger(sMsg:='Valve closed.', eSevr:=TcEventSeverity.Info);
      END_CASE
      ePreviousState := stVcnVat590.eValveControl;
  END_IF


// Log valve open
tAction(CLK:= (stVcnVat590.eValveControl = E_VCN_VAT590.OpenValve) );
IF tAction.Q THEN fbLogger(sMsg:='Valve commanded to fully open', eSevr:=TcEventSeverity.Info); END_IF
END_ACTION

ACTION ReadCoeParameters:
CASE nCaseReadCoe OF
    0:
        stVcnVat590.bCoeError := TRUE;
        IF rtCoeReset.Q THEN
            nCaseReadCoe := 1;
            stVcnVat590.bCoeError := FALSE;
            bFirstRead := TRUE; // Set bFirstRead after Coe interface reset
        END_IF
    1:
        fbCoeRead.nIndex := cPressCtrl.nIndex;
        fbCoeRead.nSubIndex := cPressCtrl.nSubIndex;
        fbCoeRead.pDstBuf := ADR(stVcnVat590.stCoeParameters.ePIDCtrl);
        fbCoeRead.cbBufLen := SIZEOF(stVcnVat590.stCoeParameters.ePIDCtrl);
        fbCoeRead.bExecute := TRUE;
    2:
        fbCoeRead.nIndex := cSensorDelay_AD.nIndex;
        fbCoeRead.nSubIndex := cSensorDelay_AD.nSubIndex;
        fbCoeRead.pDstBuf := ADR(stVcnVat590.stCoeParameters.fSensorDelay_AD);
        fbCoeRead.cbBufLen := SIZEOF(stVcnVat590.stCoeParameters.fSensorDelay_AD);
        fbCoeRead.bExecute := TRUE;
    3:
        fbCoeRead.nIndex := cRampTime_AD.nIndex;
        fbCoeRead.nSubIndex := cRampTime_AD.nSubIndex;
        fbCoeRead.pDstBuf := ADR(stVcnVat590.stCoeParameters.fRampTime_AD);
        fbCoeRead.cbBufLen := SIZEOF(stVcnVat590.stCoeParameters.fRampTime_AD);
        fbCoeRead.bExecute := TRUE;
    4:
        fbCoeRead.nIndex := cRampMode_AD.nIndex;
        fbCoeRead.nSubIndex := cRampMode_AD.nSubIndex;
        fbCoeRead.pDstBuf := ADR(stVcnVat590.stCoeParameters.bRampMode_AD);
        fbCoeRead.cbBufLen := SIZEOF(stVcnVat590.stCoeParameters.bRampMode_AD);
        fbCoeRead.bExecute := TRUE;
    5:
        fbCoeRead.nIndex := cGainFactor_AD.nIndex;
        fbCoeRead.nSubIndex := cGainFactor_AD.nSubIndex;
        fbCoeRead.pDstBuf := ADR(stVcnVat590.stCoeParameters.fGainFactor_AD);
        fbCoeRead.cbBufLen := SIZEOF(stVcnVat590.stCoeParameters.fGainFactor_AD);
        fbCoeRead.bExecute := TRUE;
    6:
        fbCoeRead.nIndex := cRampTime_FIX1.nIndex;
        fbCoeRead.nSubIndex := cRampTime_FIX1.nSubIndex;
        fbCoeRead.pDstBuf := ADR(stVcnVat590.stCoeParameters.fRampTime_FIX1);
        fbCoeRead.cbBufLen := SIZEOF(stVcnVat590.stCoeParameters.fRampTime_FIX1);
        fbCoeRead.bExecute := TRUE;
    7:
        fbCoeRead.nIndex := cRampMode_FIX1.nIndex;
        fbCoeRead.nSubIndex := cRampMode_FIX1.nSubIndex;
        fbCoeRead.pDstBuf := ADR(stVcnVat590.stCoeParameters.bRampMode_FIX1);
        fbCoeRead.cbBufLen := SIZEOF(stVcnVat590.stCoeParameters.bRampMode_FIX1);
        fbCoeRead.bExecute := TRUE;
    8:
        fbCoeRead.nIndex := cCtrlDir_FIX1.nIndex;
        fbCoeRead.nSubIndex := cCtrlDir_FIX1.nSubIndex;
        fbCoeRead.pDstBuf := ADR(stVcnVat590.stCoeParameters.bCtrlDir_FIX1);
        fbCoeRead.cbBufLen := SIZEOF(stVcnVat590.stCoeParameters.bCtrlDir_FIX1);
        fbCoeRead.bExecute := TRUE;
    9:
        fbCoeRead.nIndex := cPGain_FIX1.nIndex;
        fbCoeRead.nSubIndex := cPGain_FIX1.nSubIndex;
        fbCoeRead.pDstBuf := ADR(stVcnVat590.stCoeParameters.fPGain_FIX1);
        fbCoeRead.cbBufLen := SIZEOF(stVcnVat590.stCoeParameters.fPGain_FIX1);
        fbCoeRead.bExecute := TRUE;
    10:
        fbCoeRead.nIndex := cIGain_FIX1.nIndex;
        fbCoeRead.nSubIndex := cIGain_FIX1.nSubIndex;
        fbCoeRead.pDstBuf := ADR(stVcnVat590.stCoeParameters.fIGain_FIX1);
        fbCoeRead.cbBufLen := SIZEOF(stVcnVat590.stCoeParameters.fIGain_FIX1);
        fbCoeRead.bExecute := TRUE;
    11:
        fbCoeRead.nIndex := cRampTime_FIX2.nIndex;
        fbCoeRead.nSubIndex := cRampTime_FIX2.nSubIndex;
        fbCoeRead.pDstBuf := ADR(stVcnVat590.stCoeParameters.fRampTime_FIX2);
        fbCoeRead.cbBufLen := SIZEOF(stVcnVat590.stCoeParameters.fRampTime_FIX2);
        fbCoeRead.bExecute := TRUE;
    12:
        fbCoeRead.nIndex := cRampMode_FIX2.nIndex;
        fbCoeRead.nSubIndex := cRampMode_FIX2.nSubIndex;
        fbCoeRead.pDstBuf := ADR(stVcnVat590.stCoeParameters.bRampMode_FIX2);
        fbCoeRead.cbBufLen := SIZEOF(stVcnVat590.stCoeParameters.bRampMode_FIX2);
        fbCoeRead.bExecute := TRUE;
    13:
        fbCoeRead.nIndex := cCtrlDir_FIX2.nIndex;
        fbCoeRead.nSubIndex := cCtrlDir_FIX2.nSubIndex;
        fbCoeRead.pDstBuf := ADR(stVcnVat590.stCoeParameters.bCtrlDir_FIX2);
        fbCoeRead.cbBufLen := SIZEOF(stVcnVat590.stCoeParameters.bCtrlDir_FIX2);
        fbCoeRead.bExecute := TRUE;
    14:
        fbCoeRead.nIndex := cPGain_FIX2.nIndex;
        fbCoeRead.nSubIndex := cPGain_FIX2.nSubIndex;
        fbCoeRead.pDstBuf := ADR(stVcnVat590.stCoeParameters.fPGain_FIX2);
        fbCoeRead.cbBufLen := SIZEOF(stVcnVat590.stCoeParameters.fPGain_FIX2);
        fbCoeRead.bExecute := TRUE;
    15:
        fbCoeRead.nIndex := cIGain_FIX2.nIndex;
        fbCoeRead.nSubIndex := cIGain_FIX2.nSubIndex;
        fbCoeRead.pDstBuf := ADR(stVcnVat590.stCoeParameters.fIGain_FIX2);
        fbCoeRead.cbBufLen := SIZEOF(stVcnVat590.stCoeParameters.fIGain_FIX2);
        fbCoeRead.bExecute := TRUE;
    16:
        fbCoeRead.nIndex := cRampTime_SP.nIndex;
        fbCoeRead.nSubIndex := cRampTime_SP.nSubIndex;
        fbCoeRead.pDstBuf := ADR(stVcnVat590.stCoeParameters.fRampTime_SP);
        fbCoeRead.cbBufLen := SIZEOF(stVcnVat590.stCoeParameters.fRampTime_SP);
        fbCoeRead.bExecute := TRUE;
    17:
        fbCoeRead.nIndex := cRampMode_SP.nIndex;
        fbCoeRead.nSubIndex := cRampMode_SP.nSubIndex;
        fbCoeRead.pDstBuf := ADR(stVcnVat590.stCoeParameters.bRampMode_SP);
        fbCoeRead.cbBufLen := SIZEOF(stVcnVat590.stCoeParameters.bRampMode_SP);
        fbCoeRead.bExecute := TRUE;
    18:
        fbCoeRead.nIndex := cPGain_SP.nIndex;
        fbCoeRead.nSubIndex := cPGain_SP.nSubIndex;
        fbCoeRead.pDstBuf := ADR(stVcnVat590.stCoeParameters.fPGain_SP);
        fbCoeRead.cbBufLen := SIZEOF(stVcnVat590.stCoeParameters.fPGain_SP);
        fbCoeRead.bExecute := TRUE;
END_CASE

ftCoeReadBusy(CLK:=fbCoeRead.bBusy);
IF ftCoeReadBusy.Q THEN
    fbCoeRead.bExecute := FALSE;
    IF NOT fbCoeRead.bError THEN
        nCaseReadCoe := nCaseReadCoe + 1;
        IF nCaseReadCoe > 18 THEN
            nCaseReadCoe := 1;
            bFirstRead := FALSE; // Reset bFirstRead after successfull readout of all parameters
        END_IF
    ELSE
        nCaseReadCoe := 0; // Go to Error state
    END_IF
END_IF

fbCoeRead();
stCoeParamsInternal := stVcnVat590.stCoeParameters; //Save current values to internal structure
END_ACTION

ACTION ReadFromInput:
(*Read from EPICS*)
fUpperLimit := LIMIT(0, stVcnVat590.fPosSetLimit, 100);
fPresMaxLim := LIMIT(1.0E-10, stVcnVat590.fPresSetLimit, 1.0E-2);
fPresRbMaxLim := LIMIT(1.0E-10, stVcnVat590.fPresRdbkLimit, 1.0E-2);
fReqPos := LIMIT(0, stVcnVat590.fReqPosition, 100);
fReqPres := LIMIT(1.0E-10, stVcnVat590.fReqPressure, 1.0E-2);

(*Read from VAT valve*)
stVcnVat590.stValveStatus.eControlMode := i_eControlMode;
stVcnVat590.stValveStatus.eFatalErrors := i_eFatalError;
stVcnVat590.nRawPosition := i_nRawPosition;
stVcnVat590.nRawPressure := i_nRawPressure;
//Mapping General statuses
stVcnVat590.stValveStatus.bFieldBusDatavalid := i_stGenStatus.Bit0FieldBusDatavalid;
stVcnVat590.stValveStatus.bZeroExecuted := i_stGenStatus.Bit1ZeroExecuted;
stVcnVat590.stValveStatus.bPingPongRxBit := i_stGenStatus.Bit2PingPongRxBit;
stVcnVat590.stValveStatus.bPressureSimulation := i_stGenStatus.Bit3PressureSimulation;
stVcnVat590.stValveStatus.bPressureSPReached := i_stGenStatus.Bit4PressureSPReached;
stVcnVat590.stValveStatus.bWarningsActive := i_stGenStatus.Bit9WarningsActive;
//Read Remote status
stVcnVat590.stValveStatus.eRemoteStatus.0 := i_stGenStatus.Bit7AccessModeBit0;
stVcnVat590.stValveStatus.eRemoteStatus.1 := i_stGenStatus.Bit8AccessModeBit1;
//Mapping General warnings
stVcnVat590.stValveStatus.bServiceRequest := i_stGenWarnings.Bit0ServiceRequest;
stVcnVat590.stValveStatus.bPowerFailureBattery := i_stGenWarnings.Bit3PowerFailureBattery;
stVcnVat590.stValveStatus.bSensMeasUnitFault := i_stGenWarnings.Bit10SensMeasUnitFault;
//Mapping Extended warnings
stVcnVat590.stValveStatus.bRemoteControlNotPossible := i_stExtnWarnings.Bit0RemoteControlNotPossible;
stVcnVat590.stValveStatus.bControlModeSPNotAllowed := i_stExtnWarnings.Bit1ControlModeSPNotAllowed;
stVcnVat590.stValveStatus.bZeroDisabled := i_stExtnWarnings.Bit2ZeroDisabled;
stVcnVat590.stValveStatus.bPFODeactivated := i_stExtnWarnings.Bit3PFODeactivated;
stVcnVat590.stValveStatus.bPressureSPOutOfRange := i_stExtnWarnings.Bit5PressureSPOutOfRange;
stVcnVat590.stValveStatus.bPositionSPOutOfRange := i_stExtnWarnings.Bit6PositionSPOutOfRange;
stVcnVat590.stValveStatus.bCtrlSPOutOfRange := i_stExtnWarnings.Bit10CtrlSPOutOfRange;
stVcnVat590.stValveStatus.bGeneralCtrlSPOutOfRange := i_stExtnWarnings.Bit11GeneralCtrlSPOutOfRange;
stVcnVat590.stValveStatus.bProcDataSettingsNotvalid := i_stExtnWarnings.Bit12ProcDataSettingsNotvalid;
//Mapping WcState - Valve Ethercat Status
stVcnVat590.bValveEthCatStatus := i_bValveEthCatStatus;
END_ACTION

ACTION SetCoeInterface:
stVat590DriveRef.sNetId := F_CreateAmsNetId(i_stVat590PlcDriveRef.aNetId);
stVat590DriveRef.nSlaveAddr := i_stVat590PlcDriveRef.nSlaveAddr;
stVat590DriveRef.nDriveNo := i_stVat590PlcDriveRef.nDriveNo;
stVat590DriveRef.nDriveType := i_stVat590PlcDriveRef.nDriveType;
fbCoeRead.stDriveRef := stVat590DriveRef;
fbCoeWrite.stDriveRef := stVat590DriveRef;
END_ACTION

METHOD SetThrottle : BOOL
VAR_INPUT
    rUpperLimit	:	REAL;
END_VAR
stVcnVat590.fPosSetLimit := LIMIT(0, rUpperLimit, 100);
END_METHOD

METHOD ValveControl : BOOL
VAR_INPUT
    state : E_VCN_VAT590; // Set Control modes
END_VAR
stVcnVat590.eValveControl := state;
END_METHOD

ACTION WriteCoeParameters:
// User will change one parameter at a time so solution with ELSIF should work OK
IF stVcnVat590.bCoeError THEN
    IF rtCoeReset.Q THEN
        stVcnVat590.bCoeError := FALSE;
    END_IF;
ELSIF bFirstRead THEN
    ;//Wait until first readout of all CoE parameters is completed
ELSIF stVcnVat590.stCoeParameters.ePIDCtrl <> stCoeParamsInternal.ePIDCtrl THEN
    fbCoeWrite.nIndex := cPressCtrl.nIndex;
    fbCoeWrite.nSubIndex := cPressCtrl.nSubIndex;
    fbCoeWrite.pSrcBuf := ADR(stVcnVat590.stCoeParameters.ePIDCtrl);
    fbCoeWrite.cbBufLen := SIZEOF(stVcnVat590.stCoeParameters.ePIDCtrl);
    fbCoeWrite.bExecute := TRUE;
ELSIF stVcnVat590.stCoeParameters.fSensorDelay_AD <> stCoeParamsInternal.fSensorDelay_AD THEN
    fbCoeWrite.nIndex := cSensorDelay_AD.nIndex;
    fbCoeWrite.nSubIndex := cSensorDelay_AD.nSubIndex;
    fbCoeWrite.pSrcBuf := ADR(stVcnVat590.stCoeParameters.fSensorDelay_AD);
    fbCoeWrite.cbBufLen := SIZEOF(stVcnVat590.stCoeParameters.fSensorDelay_AD);
    fbCoeWrite.bExecute := TRUE;
ELSIF stVcnVat590.stCoeParameters.fRampTime_AD <> stCoeParamsInternal.fRampTime_AD THEN
    fbCoeWrite.nIndex := cRampTime_AD.nIndex;
    fbCoeWrite.nSubIndex := cRampTime_AD.nSubIndex;
    fbCoeWrite.pSrcBuf := ADR(stVcnVat590.stCoeParameters.fRampTime_AD);
    fbCoeWrite.cbBufLen := SIZEOF(stVcnVat590.stCoeParameters.fRampTime_AD);
    fbCoeWrite.bExecute := TRUE;
ELSIF stVcnVat590.stCoeParameters.bRampMode_AD <> stCoeParamsInternal.bRampMode_AD THEN
    fbCoeWrite.nIndex := cRampMode_AD.nIndex;
    fbCoeWrite.nSubIndex := cRampMode_AD.nSubIndex;
    fbCoeWrite.pSrcBuf := ADR(stVcnVat590.stCoeParameters.bRampMode_AD);
    fbCoeWrite.cbBufLen := SIZEOF(stVcnVat590.stCoeParameters.bRampMode_AD);
    fbCoeWrite.bExecute := TRUE;
ELSIF stVcnVat590.stCoeParameters.fGainFactor_AD <> stCoeParamsInternal.fGainFactor_AD THEN
    fbCoeWrite.nIndex := cGainFactor_AD.nIndex;
    fbCoeWrite.nSubIndex := cGainFactor_AD.nSubIndex;
    fbCoeWrite.pSrcBuf := ADR(stVcnVat590.stCoeParameters.fGainFactor_AD);
    fbCoeWrite.cbBufLen := SIZEOF(stVcnVat590.stCoeParameters.fGainFactor_AD);
    fbCoeWrite.bExecute := TRUE;
ELSIF stVcnVat590.stCoeParameters.fRampTime_FIX1 <> stCoeParamsInternal.fRampTime_FIX1 THEN
    fbCoeWrite.nIndex := cRampTime_FIX1.nIndex;
    fbCoeWrite.nSubIndex := cRampTime_FIX1.nSubIndex;
    fbCoeWrite.pSrcBuf := ADR(stVcnVat590.stCoeParameters.fRampTime_FIX1);
    fbCoeWrite.cbBufLen := SIZEOF(stVcnVat590.stCoeParameters.fRampTime_FIX1);
    fbCoeWrite.bExecute := TRUE;
ELSIF stVcnVat590.stCoeParameters.bRampMode_FIX1 <> stCoeParamsInternal.bRampMode_FIX1 THEN
    fbCoeWrite.nIndex := cRampMode_FIX1.nIndex;
    fbCoeWrite.nSubIndex := cRampMode_FIX1.nSubIndex;
    fbCoeWrite.pSrcBuf := ADR(stVcnVat590.stCoeParameters.bRampMode_FIX1);
    fbCoeWrite.cbBufLen := SIZEOF(stVcnVat590.stCoeParameters.bRampMode_FIX1);
    fbCoeWrite.bExecute := TRUE;
ELSIF stVcnVat590.stCoeParameters.bCtrlDir_FIX1 <> stCoeParamsInternal.bCtrlDir_FIX1 THEN
    fbCoeWrite.nIndex := cCtrlDir_FIX1.nIndex;
    fbCoeWrite.nSubIndex := cCtrlDir_FIX1.nSubIndex;
    fbCoeWrite.pSrcBuf := ADR(stVcnVat590.stCoeParameters.bCtrlDir_FIX1);
    fbCoeWrite.cbBufLen := SIZEOF(stVcnVat590.stCoeParameters.bCtrlDir_FIX1);
    fbCoeWrite.bExecute := TRUE;
ELSIF stVcnVat590.stCoeParameters.fPGain_FIX1 <> stCoeParamsInternal.fPGain_FIX1 THEN
    fbCoeWrite.nIndex := cPGain_FIX1.nIndex;
    fbCoeWrite.nSubIndex := cPGain_FIX1.nSubIndex;
    fbCoeWrite.pSrcBuf := ADR(stVcnVat590.stCoeParameters.fPGain_FIX1);
    fbCoeWrite.cbBufLen := SIZEOF(stVcnVat590.stCoeParameters.fPGain_FIX1);
    fbCoeWrite.bExecute := TRUE;
ELSIF stVcnVat590.stCoeParameters.fIGain_FIX1 <> stCoeParamsInternal.fIGain_FIX1 THEN
    fbCoeWrite.nIndex := cIGain_FIX1.nIndex;
    fbCoeWrite.nSubIndex := cIGain_FIX1.nSubIndex;
    fbCoeWrite.pSrcBuf := ADR(stVcnVat590.stCoeParameters.fIGain_FIX1);
    fbCoeWrite.cbBufLen := SIZEOF(stVcnVat590.stCoeParameters.fIGain_FIX1);
    fbCoeWrite.bExecute := TRUE;
ELSIF stVcnVat590.stCoeParameters.fRampTime_FIX2 <> stCoeParamsInternal.fRampTime_FIX2 THEN
    fbCoeWrite.nIndex := cRampTime_FIX2.nIndex;
    fbCoeWrite.nSubIndex := cRampTime_FIX2.nSubIndex;
    fbCoeWrite.pSrcBuf := ADR(stVcnVat590.stCoeParameters.fRampTime_FIX2);
    fbCoeWrite.cbBufLen := SIZEOF(stVcnVat590.stCoeParameters.fRampTime_FIX2);
    fbCoeWrite.bExecute := TRUE;
ELSIF stVcnVat590.stCoeParameters.bRampMode_FIX2 <> stCoeParamsInternal.bRampMode_FIX2 THEN
    fbCoeWrite.nIndex := cRampMode_FIX2.nIndex;
    fbCoeWrite.nSubIndex := cRampMode_FIX2.nSubIndex;
    fbCoeWrite.pSrcBuf := ADR(stVcnVat590.stCoeParameters.bRampMode_FIX2);
    fbCoeWrite.cbBufLen := SIZEOF(stVcnVat590.stCoeParameters.bRampMode_FIX2);
    fbCoeWrite.bExecute := TRUE;
ELSIF stVcnVat590.stCoeParameters.bCtrlDir_FIX2 <> stCoeParamsInternal.bCtrlDir_FIX2 THEN
    fbCoeWrite.nIndex := cCtrlDir_FIX2.nIndex;
    fbCoeWrite.nSubIndex := cCtrlDir_FIX2.nSubIndex;
    fbCoeWrite.pSrcBuf := ADR(stVcnVat590.stCoeParameters.bCtrlDir_FIX2);
    fbCoeWrite.cbBufLen := SIZEOF(stVcnVat590.stCoeParameters.bCtrlDir_FIX2);
    fbCoeWrite.bExecute := TRUE;
ELSIF stVcnVat590.stCoeParameters.fPGain_FIX2 <> stCoeParamsInternal.fPGain_FIX2 THEN
    fbCoeWrite.nIndex := cPGain_FIX2.nIndex;
    fbCoeWrite.nSubIndex := cPGain_FIX2.nSubIndex;
    fbCoeWrite.pSrcBuf := ADR(stVcnVat590.stCoeParameters.fPGain_FIX2);
    fbCoeWrite.cbBufLen := SIZEOF(stVcnVat590.stCoeParameters.fPGain_FIX2);
    fbCoeWrite.bExecute := TRUE;
ELSIF stVcnVat590.stCoeParameters.fIGain_FIX2 <> stCoeParamsInternal.fIGain_FIX2 THEN
    fbCoeWrite.nIndex := cIGain_FIX2.nIndex;
    fbCoeWrite.nSubIndex := cIGain_FIX2.nSubIndex;
    fbCoeWrite.pSrcBuf := ADR(stVcnVat590.stCoeParameters.fIGain_FIX2);
    fbCoeWrite.cbBufLen := SIZEOF(stVcnVat590.stCoeParameters.fIGain_FIX2);
    fbCoeWrite.bExecute := TRUE;
ELSIF stVcnVat590.stCoeParameters.fRampTime_SP <> stCoeParamsInternal.fRampTime_SP THEN
    fbCoeWrite.nIndex := cRampTime_SP.nIndex;
    fbCoeWrite.nSubIndex := cRampTime_SP.nSubIndex;
    fbCoeWrite.pSrcBuf := ADR(stVcnVat590.stCoeParameters.fRampTime_SP);
    fbCoeWrite.cbBufLen := SIZEOF(stVcnVat590.stCoeParameters.fRampTime_SP);
    fbCoeWrite.bExecute := TRUE;
ELSIF stVcnVat590.stCoeParameters.bRampMode_SP <> stCoeParamsInternal.bRampMode_SP THEN
    fbCoeWrite.nIndex := cRampMode_SP.nIndex;
    fbCoeWrite.nSubIndex := cRampMode_SP.nSubIndex;
    fbCoeWrite.pSrcBuf := ADR(stVcnVat590.stCoeParameters.bRampMode_SP);
    fbCoeWrite.cbBufLen := SIZEOF(stVcnVat590.stCoeParameters.bRampMode_SP);
    fbCoeWrite.bExecute := TRUE;
ELSIF stVcnVat590.stCoeParameters.fPGain_SP <> stCoeParamsInternal.fPGain_SP THEN
    fbCoeWrite.nIndex := cPGain_SP.nIndex;
    fbCoeWrite.nSubIndex := cPGain_SP.nSubIndex;
    fbCoeWrite.pSrcBuf := ADR(stVcnVat590.stCoeParameters.fPGain_SP);
    fbCoeWrite.cbBufLen := SIZEOF(stVcnVat590.stCoeParameters.fPGain_SP);
    fbCoeWrite.bExecute := TRUE;
END_IF

ftCoeWriteBusy(CLK:=fbCoeWrite.bBusy);
IF ftCoeWriteBusy.Q THEN
    fbCoeWrite.bExecute := FALSE;
    IF fbCoeWrite.bError THEN
        stVcnVat590.bCoeError := TRUE;
    END_IF
END_IF

fbCoeWrite();
END_ACTION

ACTION WriteToOutput:
(*Write to EPICS*)
stVcnVat590.bIlkOK := bExtIlkOK;
stVcnVat590.nPositionSP := REAL_TO_DINT(fCalcPosSP);
stVcnVat590.nPressureSP := REAL_TO_DINT(fCalcPresSP);
stVcnVat590.fReqPosition := fReqPos;
stVcnVat590.fReqPressure := fReqPres;
stVcnVat590.fPresSetLimit := fPresMaxLim;
stVcnVat590.fPosSetLimit := fUpperLimit;

(*Write to VAT valve*)
o_eCtrlModeSP := eValveModeSP;
o_nRawPositionSP := REAL_TO_DINT(fCalcPosSP);
o_nRawPressureSP := REAL_TO_DINT(fCalcPresSP);
o_stGenCtrlSP.Bit0ExecuteZero := stVcnVat590.bZero;
o_stGenCtrlSP.Bit4AccessMode := bRemAcsToggle;
END_ACTION

END_FUNCTION_BLOCK

// ---- POUs/Functions/Valves/FB_VFS_2OO3.TcPOU
(* This function block implements basic functionality for Fast Shutter/Valves*)
(* NOTE: All 3 gauge cards with fast TTL output need to be installed in the same gauge controller*)
(* Create a separate virtual PLC for the fast shutter logic, and tie/map this task to the FAST I/O portion of the ethercat bus,
 so we can scan these I/Os faster than the rest of the vacuum I/Os.
The Fast shutter was tested with PLC task Cycle Base Time 50us with cycle time 0.050ms.*)
FUNCTION_BLOCK FB_VFS_2OO3 EXTENDS FB_Valve
VAR_INPUT
    i_xPMPS_OK : BOOL; (*External MPS interlock, Set to TRUE when no PMPS interlock is required*)
    i_xExt_OK : BOOL; (*Other External Interlock, Set to True when no external interlock is required*)
    i_sDevName : T_MaxString := 'VFS'; (*Device name for diagnostic*)
    i_xVeto_Enable : BOOL := FALSE; (*Set to TRUE if there is a Veto Valve to this VFS*)
END_VAR
VAR_IN_OUT
    io_fbFFHWO : FB_HardwareFFOutput;
END_VAR
VAR
    xOPN_OK : BOOL;         //internal variable OK to Open signal
    xERR_ExtFault : BOOL;   //internal variable External Fault signal
    xVeto : BOOL;           //internal variable Veto signal
    xTrigger : BOOL;        //internal trigger signal, output of 2oo3 logic
    xPress_OK : BOOL;       //internal signal indicating if at gauges are connected and OK
    //Fault counter triggers
    rtFault_IG1 : R_TRIG;
    rtFault_IG2 : R_TRIG;
    rtFault_IG3 : R_TRIG;

    //PMPS
    fbFF : FB_FastFault :=(
        i_DevName := 'VFS',
        i_Desc := 'Fault occurs when fast valve is not in open state',
        i_TypeCode := 16#1010);

    rDiffPressAllowed : REAL := 22.5;     //Torr, Default value comes from Vat Valve Manual
    rDiffPress : REAL;                    //Current pressure

    xFirstPass : BOOL := TRUE;            //Do something on first pass, after that set to FALSE

    rtOPN_SW : R_TRIG;                    //Detect rising endge on i_xOPN_SW input

    tonDelOK : TON;
    rtOK : R_TRIG;
    tonOvrd	: TON;

    tDelOK : TIME := T#60S;
    tOvrd : TIME := T#10s;
    rTrigOverrideOpen : R_TRIG;

    xClose : BOOL;
    xOpen : BOOL;
    CloseTimer : TON;
    TimDur : TIME := T#20MS;
    OpenTimer : TON;
    OpenTimDur : TIME := T#2S;

    (*Timeouts*)
    tCLSTimeOutDuration : TIME := T#0.5S;
    tOPNTimeOutDuration : TIME := T#10S;
    tOPNtimeout : TON;
    tCLStimeout : TON;


    (*IO to the valve(s)*)
    i_xOpnLS	AT%I* : BOOL; //VFS Open limit switch input
    i_xClsLS	AT%I* : BOOL; //VFS Close limit switch input
    q_xClose_A	AT%Q* : BOOL; //3x Valve Close output signals (current req.)
    q_xClose_B	AT%Q* : BOOL; //3x Valve Close output signals (current req.)
    q_xClose_C	AT%Q* : BOOL; //3x Valve Close output signals (current req.)
    q_xOPN_DO	AT%Q* : BOOL; //Valve Open output signal
    (*3x Fast trigger Inputs from CC Gauge controller.
      Make sure all tri CC gauge cards are in the same controller*)
    i_xTriggerIG1 AT%I* : BOOL; //Fast trigger input from CC gauge 1
    i_xTriggerIG2 AT%I* : BOOL; //Fast trigger input from CC gauge 2
    i_xTriggerIG3 AT%I* : BOOL; //Fast trigger input from CC gauge 3

    (*VETO Devices*)
    i_xVetoValveOpenDO AT%I* : BOOL; (*Link to VFS Interface*)
    i_xVetoValveClosed AT%I* : BOOL; (*Link to VFS Interface*)

    (*Interface with external system*)
    i_e2OO3_MODE       AT%I* : E_2OO3_MODE; (*Link to VFS Interface, 2oo3 mode selector*)
    i_xPress_OK_IG1    AT%I* : BOOL; (*Link to VFS Interface, IG.xPRESS_OK, to make sure that the device is connected*)
    i_xPress_OK_IG2    AT%I* : BOOL; (*Link to VFS Interface, IG.xPRESS_OK, to make sure that the device is connected*)
    i_xPress_OK_IG3    AT%I* : BOOL; (*Link to VFS Interface, IG.xPRESS_OK, to make sure that the device is connected*)
    i_xOPN_SW          AT%I* : BOOL; (*Link to VFS Interface, external open signal e.g epics*)
    i_xCLS_SW          AT%I* : BOOL; (*Link to VFS Interface, external close signal e.g epics*)
    i_xVAC_FAULT_Reset AT%I* : BOOL; (*Link to VFS Interface Valve Vacuum OK, is set to False when there is Vacuum Fault*)
    i_xOverrideMode    AT%I* : BOOL; (*Link to VFS Interface, To be linked to global override bit. This Overrides Vacuum logic only, EPS, MPS and PMPS are still enforces*)
    i_xOverrideOpen    AT%I* : BOOL; (*Link to VFS Interface*)
    q_xTrigger         AT%Q* : BOOL; (*Link to VFS Interface*)
    q_xVFS_Open        AT%Q* : BOOL; (*Link to VFS Interface*)
    q_xVFS_Closed      AT%Q* : BOOL; (*Link to VFS Interface*)
    q_xVAC_FAULT_OK    AT%Q* : BOOL; (*Link to VFS Interface, Valve Vacuum OK, is set to False when there is Vacuum Fault*)
    q_xMPS_OK          AT%Q* : BOOL; (*Link to VFS Interface, MPS Fault OK, is set when the Valve is Open and there is no trigger*)
    q_eVFS_State       AT%Q* : E_VGC; (*Link to VFS Interface*)
    q_nFltCount_IG1    AT%Q* : UINT; (*Link to VFS Interface*)
    q_nFltCount_IG2    AT%Q* : UINT; (*Link to VFS Interface*)
    q_nFltCount_IG3    AT%Q* : UINT; (*Link to VFS Interface*)
END_VAR
VAR PERSISTENT
    nFaultCounter_IG1 : UINT;  //Fault counter for IG1
    nFaultCounter_IG2 : UINT;  //Fault counter for IG2
    nFaultCounter_IG3 : UINT;  //Fault counter for IG3
END_VAR

(*Fast Shutter/Valve Function Block*)
(*M.Ghaly Feb 2019*)
(*J. Govednik Jan 2022 Adding 2OO3 logic*)

(* Fast Shutters do not function as complete isolation valves, but are intended to rapidly limit conductance
between vacuum regions.  They should be installed in conjunction with isolation gate valves.  The conductance
of the fast shutter in the closed state may be sufficiently low as to create an isolated vacuum region.
Thus, at least a pirani gauge, that can measure a pressure down to 1x10-4 Torr, needs to be installed between
the shutter and the isolation gate valve.
In the case where a gauge is not installed, the neigboring gate Valves should not be opened unless the shutter
is Open.
*)

(*On first PLC pass, put valve into vented state, which implies a closed valve*)
IF xFirstPass THEN
    fbFF.i_DevName := i_sDevName;
    xFirstPass := FALSE;
END_IF

(*set Veto bit*)
IF (i_xVeto_Enable) THEN
    xVeto := (i_xVetoValveClosed AND NOT i_xVetoValveOpenDO);
    ELSE xVeto := FALSE;
END_IF

(*User will be able to select gauge channel or 2oo3 function*)
CASE i_e2OO3_MODE OF
    E_2OO3_MODE.MODE_2OO3:
        (*2oo3 logic*)
        //First let's verify that at least 2 gauges are connected
        xPress_OK := (i_xPress_OK_IG1 AND i_xPress_OK_IG2) OR
                      (i_xPress_OK_IG1 AND i_xPress_OK_IG3) OR
                      (i_xPress_OK_IG2 AND i_xPress_OK_IG3);

        //Each trigger input validated with Press OK bit which indicates if the gauge is connected or disconnected
        IF xPress_OK THEN
            xTrigger := ((i_xTriggerIG1 OR NOT i_xPress_OK_IG1) AND (i_xTriggerIG2 OR NOT i_xPress_OK_IG2)) OR
                        ((i_xTriggerIG1 OR NOT i_xPress_OK_IG1) AND (i_xTriggerIG3 OR NOT i_xPress_OK_IG3)) OR
                        ((i_xTriggerIG2 OR NOT i_xPress_OK_IG2) AND (i_xTriggerIG3 OR NOT i_xPress_OK_IG3));
            (*
            xTrigger := ((i_xTriggerIG1 AND i_xPress_OK_IG1) AND (i_xTriggerIG2 AND i_xPress_OK_IG2)) OR
                        ((i_xTriggerIG1 AND i_xPress_OK_IG1) AND (i_xTriggerIG3 AND i_xPress_OK_IG3)) OR
                        ((i_xTriggerIG2 AND i_xPress_OK_IG2) AND (i_xTriggerIG3 AND i_xPress_OK_IG3));
            *)
        ELSE
            xTrigger := TRUE;
        END_IF
    E_2OO3_MODE.IG1:
        xPress_OK := i_xPress_OK_IG1;
        xTrigger := i_xTriggerIG1 OR NOT i_xPress_OK_IG1;
    E_2OO3_MODE.IG2:
        xPress_OK := i_xPress_OK_IG2;
        xTrigger := i_xTriggerIG2 OR NOT i_xPress_OK_IG2;
    E_2OO3_MODE.IG3:
        xPress_OK := i_xPress_OK_IG3;
        xTrigger := i_xTriggerIG3 OR NOT i_xPress_OK_IG3;
END_CASE;

//xVeto:= i_xVeto AND (i_xVetoValveClosed AND NOT i_xVetoValveOpenDO);
(*Input Trigger to close the Fast Shutter*)
(*Neighboring Valves Should also be triggered to Close*)
//IF ((xTrigger) OR NOT (i_xPress_OK) OR NOT (i_xExt_OK))  AND NOT (xVeto) AND NOT (tonOvrd.Q AND i_xOverrideMode) THEN
IF ((xTrigger) OR NOT (i_xExt_OK))  AND NOT (xVeto) AND NOT (tonOvrd.Q AND i_xOverrideMode) THEN
    xClose := TRUE;
    xOpen := FALSE;
    q_xVAC_FAULT_OK := FALSE;
    xERR_ExtFault := TRUE;
    i_xCLS_SW := TRUE;
    q_xOPN_DO := FALSE;
    //i_xOPN_SW :=FALSE;
ELSIF (i_xCLS_SW) THEN
    xClose := TRUE;
    xOpen := FALSE;
    q_xVAC_FAULT_OK:= FALSE;
    i_xCLS_SW := TRUE;
    q_xOPN_DO := FALSE;
    //i_xOPN_SW :=FALSE;
ELSIF ((rtOPN_SW.Q) AND xOPN_OK AND NOT i_xOpnLS) OR (tonOvrd.Q AND i_xOverrideMode) THEN
    q_xOPN_DO := TRUE;
END_IF

//Hold Valve close signals to TRUE until limit swith is hit
IF (xClose) AND (NOT i_xClsLS) THEN
    q_xClose_A := TRUE;
    q_xClose_B := TRUE;
    q_xClose_C := TRUE;
END_IF

//Set Valve close signals to FALSE when close timer expires or close limit switch is closed
IF(CloseTimer.Q) OR (i_xClsLS) THEN
    q_xClose_A := FALSE;
    q_xClose_B := FALSE;
    q_xClose_C := FALSE;
    xClose := FALSE;
    //i_xOPN_SW := FALSE;
END_IF

//Set Valve open signal to FALSE when open timer expires or open limit switch is closed
IF(OpenTimer.Q) AND (i_xOpnLS) THEN
    q_xOPN_DO :=  FALSE;
    i_xOPN_SW := FALSE;
    xOpen := FALSE;
END_IF

(*Neighboring Valves Interlock bit is reset When the Vacuum event error is reset and the Shutter is opened*)
IF ((NOT xTrigger) OR xVeto) AND (NOT xERR_ExtFault) AND i_xOpnLS THEN
    q_xVAC_FAULT_OK := TRUE;
END_IF

(*OPN OK evaluation bit*)
xOPN_OK := (NOT xERR_ExtFault) AND (NOT xTrigger OR xVeto) ;

(*When the valve  is open MPS is OK*)
//q_xMPS_OK := i_xOpnLS AND ((NOT xTrigger AND i_xPress_OK) OR xVeto)  AND NOT(i_xCLS_SW);
q_xMPS_OK := i_xOpnLS AND (NOT xTrigger OR xVeto) AND NOT(i_xCLS_SW);


(*Override logic*)
(*Goal: give ability to override, but do so in a way that people won't forget it.
Solution: Override only after ten seconds of override, protect against blips,
when the valve permission goes true for more than ten seconds consistently, remove override
*)
rTrigOverrideOpen (CLK := i_xOverrideOpen); // Not used

tonDelOK (IN := xOPN_OK, PT := tDelOK);
rtOK (CLK := tonDelOK.Q);

IF rtOK.Q AND i_xOverrideOpen THEN
    i_xOverrideOpen := FALSE;
    //if (i_xOpnLS) AND (i_xOverrideMode) THEN i_xOPN_SW := TRUE; END_IF //for seamless transition
    //Log
    fbLogger(sMsg := 'Override expired', eSevr := TcEventSeverity.Warning);
END_IF

//Override timer
tonOvrd(IN := i_xOverrideOpen, PT := tOvrd);


//Assign valve state
IF (xTrigger) THEN
    q_eVFS_State := E_VGC.Triggered;
ELSIF xERR_ExtFault THEN
    q_eVFS_State :=  E_VGC.Vac_Fault;
ELSIF NOT i_xClsLS AND tCLStimeout.Q THEN
    q_eVFS_State :=  E_VGC.Cls_Timeout;
ELSIF NOT i_xOpnLS AND tOPNtimeout.Q THEN
    q_eVFS_State :=  E_VGC.Opn_Timeout;
ELSE
    q_eVFS_State :=  E_VGC.At_Vac;
END_IF

(*Timers*)
CloseTimer (IN := xClose, PT := TimDur);
OpenTimer (IN := i_xOpnLS, PT := OpenTimDur);
tOPNtimeout (IN := q_xOPN_DO, PT := tOPNTimeOutDuration);
tCLStimeout (IN := q_xClose_A, PT := tCLSTimeOutDuration);

//Detecting rising edge for i_xOPN_SW (epics command)
rtOPN_SW (CLK := i_xOPN_SW);

(*Gauge fault counters*)
//IG1
rtFault_IG1(CLK := i_xTriggerIG1 AND NOT xTrigger);
IF rtFault_IG1.Q THEN
    nFaultCounter_IG1 := nFaultCounter_IG1 + 1;
END_IF
//IG2
rtFault_IG2(CLK := i_xTriggerIG2 AND NOT xTrigger);
IF rtFault_IG2.Q THEN
    nFaultCounter_IG2 := nFaultCounter_IG2 + 1;
END_IF
//IG3
rtFault_IG3(CLK := i_xTriggerIG3 AND NOT xTrigger);
IF rtFault_IG3.Q THEN
    nFaultCounter_IG3 := nFaultCounter_IG3 + 1;
END_IF

(*Soft IO Mapping*)
IO();

(*Alarm reset *)
ACT_ResetAlarms();

(*FAST FAULT*)
fbFF(i_xOK := q_xMPS_OK,
    i_xReset := i_xVAC_FAULT_Reset,
    i_xAutoReset := TRUE,
    io_fbFFHWO := io_fbFFHWO);

ACTION ACT_ResetAlarms:
//iq_stValve.xERR_DifPres R= i_xResetFault;

//iq_stValve.bErrorPresent R= i_xResetFault;

IF (NOT xTrigger AND xPress_OK AND i_xVAC_FAULT_Reset) OR xVeto THEN
    xERR_ExtFault := FALSE;
    i_xVAC_FAULT_Reset := FALSE;
END_IF


IF (xTrigger OR NOT xPress_OK) AND NOT xVeto THEN
    i_xVAC_FAULT_Reset := FALSE;
END_IF
END_ACTION

ACTION IO:
q_xTrigger := xTrigger;
q_xVFS_Closed := i_xClsLS;
q_xVFS_Open := i_xOpnLS;

q_nFltCount_IG1 := nFaultCounter_IG1;
q_nFltCount_IG2 := nFaultCounter_IG2;
q_nFltCount_IG3 := nFaultCounter_IG3;
END_ACTION

END_FUNCTION_BLOCK

// ---- POUs/Functions/Valves/FB_VGC_NEW.TcPOU
(* This function block implements basic functionality for Isolation Gate Valves*)
(* This function block interlock is as follows:
1. The valve can be opened when the pressures on both sides is
below than the pressure setpoint.
2. This rule persists until the interlock is overrided.
3. Once at-vac, the valve will close if the pressure on either side rises above the hysteresis pressure *)
(*This function block also implements EPS interlocks and Fast MPS trigger*)
{attribute 'no_check'}
{attribute 'reflection'}
FUNCTION_BLOCK FB_VGC_NEW Extends FB_Valve
VAR_IN_OUT

END_VAR

VAR_INPUT
    (*Upstream Gauge, usually ion gauge*)
    i_stUSG	:	ST_VG;
    (*Downstream Gauge, usually ion gauge*)
    i_stDSG	:	ST_VG;
    {attribute 'pytmc' := '
    pv: Dis_DPIlk
    '}
    i_xDis_DPIlk : BOOL := FALSE;  (* Set to true when calling the function to disable the differential pressure interlock *)

    {attribute 'pytmc' := '
    pv: EPS_OK
    '}
    i_xEPS_OK:	BOOL	:= TRUE; (*External EPS interlock, Set to TRUE when no EPS interlock is required, otherwise set to correct interlock signal*)
    i_xExt_OK: BOOL; (*Other External Interlock, Set to True when no external interlock is required. If this Valve is neigboring a Fast Shutter this should be linked to the fast shutter xVAC_FAULT_OK*)
    i_xOverrideMode : BOOL; (*To be linked to global override bit. This Overrides Vacuum logic only, EPS, MPS and PMPS are still enforces*)
    // Reset fault
    {attribute 'pytmc' := '
    pv: FF_Reset
    '}
    i_xReset: BOOL;
    i_xIsAperture:BOOL :=FALSE; // Set tp True if this is an Aperture Valve, the MPS Fault will trip only when moving.
    i_sDevName : T_MaxString :=  'VGC'; // Device name for diagnostic

END_VAR

VAR_OUTPUT
    {attribute 'pytmc' := '
    pv:
    '}
    iq_stValve : ST_VGC; (* All valve data and states will be in this struct*)

    {attribute 'pytmc' := '
    pv: MPS_FAULT_OK
    field: ZNAM MPS FAULT ;
    field: ONAM MPS OK ;
    '}
    xMPS_OK:	BOOL; (*MPS Fast OK, is set when the Valve is Open*)

    {attribute 'pytmc' := '
    pv: OVRD_Countdown
    field: EGU HOUR;
    '}
    tOvrd_countdown : LREAL; (* Countdown of the valve overriding in hour*)
END_VAR

VAR_IN_OUT
    io_fbFFHWO    :    FB_HardwareFFOutput;
END_VAR

VAR
    FFO    :    FB_FastFault :=(
        i_Desc := 'Fault occurs when the valve is not in open state',
        i_TypeCode := 16#1010);

    {attribute 'instance-path'}
    {attribute 'noinit'}
    sPath: STRING;

    rDiffPressAllowed	:	REAL := 22.5; // Torr, Default value comes from Vat Valve Manual
    rDiffPress : REAL;
    set : BOOL;
    reset: BOOL;

    xFirstPass	:	BOOL;
    fbFSInit		:	R_TRIG;

    tonOvrdExpired : TON;
    rtOK	:	R_TRIG;
    tonOvrd	:	TON;
    rtOpen	:	R_TRIG;
    ftClose: F_TRIG;

    {attribute 'pytmc' := '
    pv: OVRD_DURATION
    io: io
    '}
    nOvrdDurationHour : REAL := 0.5;
    OvrdHrFix : REAL;
    tOvrdDurationMS : TIME;

//    tDelOK	:	TIME := T#60S;
    tOvrd	:	TIME := T#10S;


    (* Timeouts*)
    tTimeOutDuration: TIME:= T#30S;
    tOPNtimeout: TON;
    tCLStimeout:TON;

    (* Timedelay on set/reset At_vac state *)
    tonSet : TON;
    tSet : TIME := T#50MS;
    tonReset : TON;
    tReset : TIME := T#50MS;


    (*IO*)
    i_xOpnLS	AT%I*: BOOL;
    i_xClsLS	AT%I*: BOOL;
    q_xOPN_DO	AT%Q*: BOOL;

    // For logging
    eVGCPrevState : E_VGC;

    rHYS_fix : REAL;
	
   //For gauge spike testing, remove before release lib
   {attribute 'pytmc' := '
    pv: GaugeSpiked
    '}
	bSpiked: BOOL;
	setSpike: BOOL;
	resetSpike: BOOL;
	tof_reset : TOF;
	sr_SR : SR;
	
END_VAR

VAR PERSISTENT
    rAT_VAC_SP	:	REAL;
    rAT_VAC_HYS :   REAL;
END_VAR

(* Vacuum gate valve
Modified from A. Wallace's VGC function
16-10-29
*)
(* 10/1/2018 Margaret Ghaly included EPS, PMPS Checkes and MPS trigger signals*)
(* 6/26/2026 Jing removed the PMPS checks, added a 50 ms delay to filter transient pressure spikes, and modified the override open function to latch for a user-configurable duration of up to 12 hours. *)


fbFSInit( CLK := TRUE, Q => xFirstPass);
(*IO Mapping*)
ACT_IO();

(* On first PLC pass, put valve into vented state, which implies a closed valve *)
IF xFirstPass THEN
    iq_stValve.eVGC_State := Vented;
    iq_stValve.pv_xOPN_SW := FALSE;
    FFO.i_DevName := i_sDevName;
    iq_stValve.sDevName := i_sDevName;
END_IF


///Check valve position
IF iq_stValve.i_xClsLS AND  iq_stValve.i_xOpnLS THEN
    iq_stValve.eState:=INVALID;
ELSIF NOT iq_stValve.i_xClsLS AND iq_stValve.i_xOpnLS AND iq_stValve.q_xOPN_DO THEN
    iq_stValve.eState:=OPEN;
ELSIF NOT iq_stValve.i_xClsLS AND iq_stValve.i_xOpnLS AND NOT iq_stValve.q_xOPN_DO THEN
    iq_stValve.eState:=OPEN_F;
ELSIF iq_stValve.i_xClsLS AND NOT iq_stValve.i_xOpnLS AND NOT iq_stValve.q_xOPN_DO THEN
    iq_stValve.eState:=CLOSED;
ELSIF NOT iq_stValve.i_xClsLS AND NOT iq_stValve.i_xOpnLS THEN
    iq_stValve.eState:=MOVING;
ELSE
    iq_stValve.eState:=INVALID;
END_IF

// Check the setpoint and hysteresis pressure from user inputs
// Hysteresis pressures should be above the setpoint and not higher than 20% of the setpoint
IF iq_stValve.rAT_VAC_SP = 0.0 THEN
    iq_stValve.rAT_VAC_SP := 0.0000001;
END_IF
rHYS_fix := LIMIT(iq_stValve.rAT_VAC_SP, iq_stValve.rAT_VAC_HYS, iq_stValve.rAT_VAC_SP*1.2);
iq_stValve.rAT_VAC_HYS := rHYS_fix;

// Valve at vacuum check
// set and rest have to latch for 50ms before change At_vac state
    set := i_stUSG.rPRESS < iq_stValve.rAT_VAC_SP AND i_stDSG.rPRESS < iq_stValve.rAT_VAC_SP AND i_stUSG.xPRESS_OK AND i_stDSG.xPRESS_OK;
    tonSet(IN:=set, PT:=tSet);
    iq_stValve.xAT_VAC S= tonSet.Q;
    reset := i_stUSG.rPRESS > iq_stValve.rAT_VAC_HYS OR i_stDSG.rPRESS > iq_stValve.rAT_VAC_HYS OR NOT i_stUSG.xPRESS_OK OR NOT i_stDSG.xPRESS_OK;
    tonReset(IN:=reset, PT:=tReset);
    iq_stValve.xAT_VAC R= tonReset.Q;
	
//Record the spikes
   setSpike := reset;
   tof_reset(IN:= reset,PT:=T#1S);//latch for 1s for EPICS Archiver
   resetSpike := tof_reset.Q;   
   sr_SR(SET1:=setSpike,RESET:=resetSpike);
   bSpiked :=sr_SR.Q1; 

// Differential pressure check
    (* Calc the differential pressure across the valve *)
    rDiffPress := ABS(i_stUSG.rPRESS - i_stDSG.rPRESS);

    (* As long as the differential pressure is less than 22.5 Torr, the valve is allowed to open *)
    IF rDiffPress <= rDiffPressAllowed AND i_stUSG.xPRESS_OK AND i_stDSG.xPRESS_OK THEN
        iq_stValve.xDP_OK := TRUE;
    ELSE
        iq_stValve.xDP_OK	:= FALSE;
        (* If the differential pressure is exceeded, even when the valve is open,
        the state is unexpected and triggers a fault, because it suggests that something
        is wrong with the valve, or gauges or mapping or there is a major leak on one side.*)
        iq_stValve.eVGC_State := ERR_DiffPress;
        iq_stValve.xERR_DifPres := TRUE;
    END_IF

// Valve state
///////////////////////////////////////////////////
CASE iq_stValve.eVGC_State OF
    Vented: (* The Vented state is used during pump down *)
        (* Assuming the pump down went well, we are now at vacuum on both sides,
        so we move to the vacuum state, otherwise remain in the vented state *)
        IF iq_stValve.xAT_VAC AND (NOT (iq_stValve.xERR_DifPres)) AND (NOT (iq_stValve.xERR_SP)) AND (NOT (iq_stValve.xERR_ExtFault))THEN
            iq_stValve.eVGC_State := AtVacuum;
        ELSE
            iq_stValve.eVGC_State := Vented;
        END_IF

    AtVacuum:
        IF iq_stValve.xAT_VAC THEN
        (* If both pressure setpoints are made,
        then enable the differential pressure interlock, regardless of the valve state
        assuming we're using some kind of ion gauge where a pressure setpoint cannot be higher than 1E-4 T *)
        iq_stValve.eVGC_State := AtVacuum;

        ELSE

            (* If the valve is open (or in an unknown state) and either gauge is not at it's vacuum setpoint,
            we have a loss of vacuum error *)
            IF (iq_stValve.i_xOpnLS OR (NOT iq_stValve.i_xOpnLS AND NOT iq_stValve.i_xClsLS)) THEN
                iq_stValve.eVGC_State := ERR_LostVac;
                iq_stValve.xERR_SP := TRUE; //TAW changed this to the ERR_SP bool because I think that's what it was intended to be?

            (* Alternatively, if the valve is already closed and we lose pressure on one side,
            it was probably intentional venting, so we calmly move back to venting mode, and
            disable the differential pressure interlock *) //??
            ELSIF iq_stValve.i_xClsLS THEN
                iq_stValve.eVGC_State := Vented;
            END_IF

        END_IF

    ERR_DiffPress:
        IF NOT (iq_stValve.xERR_DifPres) THEN
            IF iq_stValve.xAT_VAC AND (NOT (iq_stValve.xERR_DifPres)) AND (NOT (iq_stValve.xERR_SP)) AND (NOT (iq_stValve.xERR_ExtFault))THEN
                iq_stValve.eVGC_State := AtVacuum;
            ELSE
                iq_stValve.eVGC_State := Vented;
            END_IF
        END_IF


    ERR_LostVac:
        IF NOT (iq_stValve.xERR_SP) THEN
            IF iq_stValve.xAT_VAC AND (NOT (iq_stValve.xERR_DifPres)) AND (NOT (iq_stValve.xERR_SP)) AND (NOT (iq_stValve.xERR_ExtFault))THEN
                iq_stValve.eVGC_State := AtVacuum;
            ELSE
                iq_stValve.eVGC_State := Vented;
            END_IF
        END_IF

    ERR_ExtFault:
        IF NOT (iq_stValve.xERR_ExtFault) AND (i_xExt_OK) THEN
            IF iq_stValve.xAT_VAC AND (NOT (iq_stValve.xERR_DifPres)) AND (NOT (iq_stValve.xERR_SP)) AND (NOT (iq_stValve.xERR_ExtFault))THEN
                iq_stValve.eVGC_State := AtVacuum;
            ELSE
                iq_stValve.eVGC_State := Vented;
            END_IF
        END_IF
END_CASE

IF (NOT i_xExt_OK) AND (iq_stValve.eState=OPEN)  THEN
    iq_stValve.eVGC_State := ERR_ExtFault;
    iq_stValve.xERR_ExtFault := TRUE;
END_IF

// Interlock evaluation - with bypass for DP ILK bypass
///////////////////////////////////////////////
IF i_xDis_DPIlk THEN
    iq_stValve.xOPN_OK := iq_stValve.xEXT_OK; // AND iq_stValve.xDP_OK ;
ELSE
    iq_stValve.xOPN_OK := iq_stValve.xEXT_OK AND iq_stValve.xAT_VAC;
END_IF


(* Valve operation *)

(* Override logic *)
(* Goal: give ability to override, but do so in a way that people won't forget it.
Solution: Override only after ten seconds of override, protect against blips,
Latch override for user defined duration and up to 12 hours. Maximum 12 hours override duration is requested by CDSO.
*)

OvrdHrFix := LIMIT (0.25,nOvrdDurationHour,12); // ensure the override hours from user input are within 0.25 hour to 12 hours (Max 12 hours required by Patrick Oppermann)
tOvrdDurationMS := DINT_TO_TIME(
                        REAL_TO_DINT (OvrdHrFix*60*60*1000.0)
                   ); //convert to time in msec

tonOvrdExpired(IN:=iq_stValve.pv_xOvrdOpn, PT:=tOvrdDurationMS);
tOvrd_countdown := TIME_TO_LREAL(tonOvrdExpired.ET)/1000.0/60/60; // remaining time in hours

IF tonOvrdExpired.Q AND iq_stValve.pv_xOvrdOpn THEN
    iq_stValve.pv_xOvrdOpn :=FALSE;
    if (iq_stValve.eState = OPEN) AND (i_xOverrideMode) THEN iq_stValve.pv_xOPN_SW := TRUE; END_IF //for seamless transition
    //Log
    fbLogger(sMsg:='Override expired', eSevr:=TcEventSeverity.Warning);
END_IF
// Release the Force Open bit when the system override is false
IF NOT (i_xOverrideMode) THEN  iq_stValve.pv_xOvrdOpn :=FALSE; END_IF
//Override timer
tonOvrd(IN:=iq_stValve.pv_xOvrdOpn, PT:=tOvrd);


(* Valve operation *)
(* Here's where we evaluate sw actions and operate the valve *)
(* Valve operation *)

ftClose(CLK:= iq_stValve.pv_xOPN_SW);
rtOpen(CLK:= iq_stValve.pv_xOPN_SW);


IF NOT (iq_stValve.xOPN_OK) THEN
    iq_stValve.pv_xOPN_SW:= FALSE; // Reset switch after interlock is lost
    IF (tonOvrd.Q AND i_xOverrideMode) THEN
        iq_stValve.pv_xOPN_SW:= TRUE; //set switch to true if valve is overrided open
    END_IF
END_IF
iq_stValve.q_xOPN_DO := (iq_stValve.pv_xOPN_SW  AND iq_stValve.xOPN_OK) OR (tonOvrd.Q AND i_xOverrideMode);



(*MPS Fault setting*)
If (i_xIsAperture ) THEN
    (* When the valve  is open or in Closed position MPS is OK, Fault while moving*)
    xMPS_OK := (i_xOpnLS  AND q_xOPN_DO) XOR (i_xClsLS  AND NOT q_xOPN_DO);
ELSE
    (* When the valve  is open MPS is OK*)
    xMPS_OK := i_xOpnLS AND NOT i_xClsLS AND q_xOPN_DO;
END_IF


///Check valve moving postion timout
IF NOT iq_stValve.i_xClsLS AND tCLStimeout.Q THEN
    iq_stValve.bErrorPresent := TRUE;
    iq_stValve.sErrorMessage := 'Close Timeout';
ELSIF NOT iq_stValve.i_xOpnLS AND tOPNtimeout.Q THEN
    iq_stValve.bErrorPresent := TRUE;
    iq_stValve.sErrorMessage := 'Open Timeout';
END_IF
IF (iq_stValve.eState=INVALID) THEN
    iq_stValve.bErrorPresent := TRUE;
    iq_stValve.sErrorMessage := CONCAT(sPath,'Invalid Valve Position');
END_IF


(*Timers*)
tOPNtimeout(IN:= iq_stValve.q_xOPN_DO, PT := tTimeOutDuration );
tCLStimeout(IN:= NOT iq_stValve.q_xOPN_DO, PT := tTimeOutDuration);


// Alarm reset
//////////////////////////////////////
ACT_ResetAlarms();

(*IO Mapping*)
ACT_IO();

// Log States and triggers
ACT_Logger();

(*Load or save the persistent variables*)
ACT_Persistent();


(*FAST FAULT*)
FFO(i_xOK := xMPS_OK,
    i_xReset := i_xReset,
    i_xAutoReset :=TRUE,
    i_DevName := i_sDevName,
    io_fbFFHWO := io_fbFFHWO);

ACTION ACT_IO:
(*inputs*)
iq_stValve.i_xOpnLS := 	i_xOpnLS;
iq_stValve.i_xClsLS:=	i_xClsLS;
iq_stValve.xEXT_OK := i_xEXT_OK;
iq_stValve.xOverrideMode := i_xOverrideMode;
(*outputs*)
q_xOPN_DO:= iq_stValve.q_xOPN_DO;

(*ILK Devices*)
iq_stValve.sIlkUSDeviceName := This^.i_stUSG.sPath;
iq_stValve.sIlkDSDeviceName := This^.i_stDSG.sPath;
END_ACTION

ACTION ACT_Logger:
// ILK logger

IF NOT (iq_stValve.xOPN_OK) AND (ePrevState = OPEN) AND NOT (TonOvrd.Q) THEN
         fbLogger(sMsg:='Lost interlock ok bit while valve was open.', eSevr:=TcEventSeverity.Critical);
END_IF


//Positiong STATE Logger
IF ePrevState <> iq_stValve.eState THEN
      CASE iq_stValve.eState OF
        INVALID:
            fbLogger(sMsg:='Valve invalid position.', eSevr:=TcEventSeverity.Critical);
          MOVING:
            fbLogger(sMsg:='Valve moving', eSevr:=TcEventSeverity.Warning);
        OPEN:
            fbLogger(sMsg:='Valve Open.', eSevr:=TcEventSeverity.Info);
        OPEN_F:
            fbLogger(sMsg:='Valve Open.', eSevr:=TcEventSeverity.Info);
        CLOSED:
            fbLogger(sMsg:='Valve closed.', eSevr:=TcEventSeverity.Info);
      END_CASE
      ePrevState := iq_stValve.eState;
  END_IF

 //Pressure STATE Logger
IF eVGCPrevState <> iq_stValve.eVGC_State THEN
      CASE iq_stValve.eVGC_State OF
        Vented:
             fbLogger(sMsg:='Vented', eSevr:=TcEventSeverity.Info);
          AtVacuum:
             fbLogger(sMsg:='Vacuum setpoint satisfied', eSevr:=TcEventSeverity.Info);
        ERR_DiffPress:
             fbLogger(sMsg:='Potential accidental vent.', eSevr:=TcEventSeverity.Critical);
        ERR_LostVac:
            fbLogger(sMsg:='Unexpected loss of vacuum while valve was open or moving.', eSevr:=TcEventSeverity.Critical);
        ERR_ExtFault:
             fbLogger(sMsg:='Lost external interlock while valve was open.', eSevr:=TcEventSeverity.Critical);
      END_CASE
      eVGCPrevState := iq_stValve.eVGC_State;
  END_IF



// Log valve timeouts
tErrorPresent(CLK:=iq_stValve.bErrorPresent);
IF tErrorPresent.Q THEN fbLogger(sMsg:=iq_stValve.sErrorMessage, eSevr:=TcEventSeverity.Warning); END_IF

// Log valve open
tAction(CLK:= iq_stValve.q_xOPN_DO);
IF tAction.Q THEN fbLogger(sMsg:='Valve commanded open', eSevr:=TcEventSeverity.Info); END_IF

// Log override mode enabled
tOverrideActivated(CLK:= (tonOvrd.Q AND i_xOverrideMode));
IF tOverrideActivated.Q THEN fbLogger(sMsg:='Valve override mode activated', eSevr:=TcEventSeverity.Warning); END_IF
END_ACTION

ACTION ACT_Persistent:
(*On first PLC pass, load the persistent value into the structrue variable*)
IF (SUPER^.bRestorePersistentData) THEN
    SUPER^.bRestorePersistentData	:= FALSE;
    IF (rAT_VAC_SP <> 0) THEN
        iq_stValve.rAT_VAC_SP := rAT_VAC_SP;
    END_IF;
    IF (rAT_VAC_HYS <> 0) THEN
            iq_stValve.rAT_VAC_HYS := rAT_VAC_HYS;
    END_IF;
END_IF
(*Check if a new value has been written in the structure variable copy it to the persistent variable*)
IF NOT (iq_stValve.rAT_VAC_SP = rAT_VAC_SP) THEN
    rAT_VAC_SP :=iq_stValve.rAT_VAC_SP;
END_IF;

IF NOT (iq_stValve.rAT_VAC_HYS = rAT_VAC_HYS) THEN
    rAT_VAC_HYS:= iq_stValve.rAT_VAC_HYS;
END_IF;
END_ACTION

ACTION ACT_ResetAlarms:
iq_stValve.xERR_DifPres R= iq_stValve.pv_xAlmRst;
iq_stValve.xERR_SP R= iq_stValve.pv_xAlmRst;
iq_stValve.bErrorPresent R= iq_stValve.pv_xAlmRst;
iq_stValve.xERR_ExtFault R= iq_stValve.pv_xAlmRst;

IF ( iq_stValve.pv_xAlmRst) THEN
    iq_stValve.sErrorMessage :='';
     iq_stValve.pv_xAlmRst := FALSE;
END_IF
END_ACTION

METHOD PUBLIC M_IsClosed : BOOL
VAR_INPUT
END_VAR
M_IsClosed := (This^.iq_stValve.eState = E_ValvePositionState.CLOSED);
END_METHOD

METHOD PUBLIC M_IsOpen : BOOL
VAR_INPUT
END_VAR
M_IsOpen := (This^.iq_stValve.eState = E_ValvePositionState.OPEN);
END_METHOD

// Use this Methode to Open or close the valve by setting the OPN_SW to the input value.
METHOD PUBLIC M_Set_OPN_SW : BOOL
VAR_INPUT
        value:BOOL;
END_VAR
This^.iq_stValve.pv_xOPN_SW := value;
END_METHOD

METHOD PUBLIC M_SetAtVacSP
VAR_INPUT
    i_fAtVacSP : REAL;
END_VAR
iq_stValve.rAT_VAC_SP := i_fAtVacSP;
END_METHOD

METHOD PUBLIC M_SetAtVacSPHys
VAR_INPUT
    i_fAtVacSPHys : REAL;
END_VAR
iq_stValve.rAT_VAC_HYS := i_fAtVacSPHys;
END_METHOD

END_FUNCTION_BLOCK

// ---- POUs/Functions/Valves/Interfaces/FB_VFS_2OO3Interface.TcPOU
(*Used as soft IO mapping to create a psuedo valve to communicate over two task on the same PLC.*)
(*NOTE: All 3 gauge cards with fast TTL output need to be installed in the same gauge controller*)
(*For FAST shutter control*)
FUNCTION_BLOCK FB_VFS_2OO3Interface EXTENDS FB_Valve
VAR_INPUT
    (*Make sure all three CC gauge cards are in the same controller*)
    IG1 : ST_VG; // The MKS422 Cold Cathode Data Structure for CC gauge 1
    IG2 : ST_VG; // The MKS422 Cold Cathode Data Structure for CC gauge 2
    IG3 : ST_VG; // The MKS422 Cold Cathode Data Structure for CC gauge 3
    Veto_Valve : ST_VGC; // The VGC structure for the Veto Valve
    {attribute 'pytmc' := '
        pv: VFS_2OO3_MODE
        io: io
    '}
    i_e2OO3_MODE : E_2OO3_MODE; // 2oo3 mode selector as EPICS Command or Input for global variable
END_VAR
VAR_OUTPUT
    {attribute 'pytmc' := '
        pv: ;
    '}
    iq_stValve : ST_VFS; (* All valve data and states will be in this struct*)
    i_xVAC_FAULT_OK AT%I* : BOOL; (*Valve Vacuum OK, is set to False when there is Vacuum Fault*)
END_VAR
VAR
    rtTriggerVetoed : R_TRIG;
    rtTriggered : R_TRIG;
    tonOvrd	: TON;
    tOvrd : TIME := T#10s;
    rtOK : R_TRIG;
    tonDelOK : TON;
    xOPN_OK : BOOL;
    tDelOK	: TIME := T#60S;
    xPress_OK : BOOL;                      //internal signal indicating if at gauges are connected and OK

    (*outputs*)
    q_e2OO3_MODE AT%Q* : E_2OO3_MODE;             //2oo3 mode selector
    q_xPRESS_OK_IG1 AT%Q* : BOOL;
    q_xPRESS_OK_IG2 AT%Q* : BOOL;
    q_xPRESS_OK_IG3 AT%Q* : BOOL;
    q_xOPN_SW AT%Q* : BOOL;
    q_xCLS_SW AT%Q* : BOOL; (*external open signal e.g epics*)
    q_xVAC_FAULT_Reset AT%Q* : BOOL; (*Valve Vacuum OK, is set to False when there is Vacuum Fault*)
    q_xOverrideMode AT%Q* : BOOL; (*To be linked to global override bit. This Overrides Vacuum logic only, EPS, MPS and PMPS are still enforces*)
    q_xOverrideOpen AT%Q* : BOOL;

    (*VETO Devices*)
    q_xVetoValveOpenDO AT%Q* : BOOL;
    q_xVetoValveClosed AT%Q* : BOOL;
    (*inputs*)
    i_xTrigger AT%I* : BOOL;
    i_xVFS_Open AT%I* : BOOL;
    i_xVFS_Closed AT%I* : BOOL;
    {attribute 'pytmc' := '
        pv: MPS_FAULT_OK
        field: ZNAM MPS FAULT ;
        field: ONAM MPS OK ;
        io: i ;
    '}
    i_xMPS_OK AT%I* : BOOL;(*MPS Fault OK, is set when the Valve is Open and there is no trigger*)
    i_eVFS_State AT%I* : E_VGC; (*Interface*)
    {attribute 'pytmc' := '
        pv: FLT_COUNT_IG1
        io: i
    '}
    i_nFltCount_IG1 AT%I* : UINT;      //Fault counter for IG1
    {attribute 'pytmc' := '
        pv: FLT_COUNT_IG2
        io: i
    '}
    i_nFltCount_IG2 AT%I* : UINT;      //Fault counter for IG2
    {attribute 'pytmc' := '
        pv: FLT_COUNT_IG3
        io: i
    '}
    i_nFltCount_IG3 AT%I* : UINT;      //Fault counter for IG3
END_VAR

(*Soft IO Mapping*)
q_xPRESS_OK_IG1 := IG1.xPRESS_OK;
q_xPRESS_OK_IG2 := IG2.xPRESS_OK;
q_xPRESS_OK_IG3 := IG3.xPRESS_OK;

(*Soft IO Mapping*)
IO();

//Check valve postion
IF iq_stValve.i_xClsLS AND  iq_stValve.i_xOpnLS THEN
    iq_stValve.eState:=INVALID;
ELSIF NOT iq_stValve.i_xClsLS AND iq_stValve.i_xOpnLS THEN
    iq_stValve.eState:=OPEN;
ELSIF iq_stValve.i_xClsLS AND NOT iq_stValve.i_xOpnLS THEN
    iq_stValve.eState:=CLOSED;
ELSIF NOT iq_stValve.i_xClsLS AND NOT iq_stValve.i_xOpnLS THEN
    iq_stValve.eState:=MOVING;
ELSE
    iq_stValve.eState:=INVALID;
END_IF
//Override timer
tonOvrd(IN:=q_xOverrideOpen, PT:=tOvrd);
tonDelOK(IN:=xOPN_OK, PT:=tDelOK);
rtOK(CLK:=tonDelOK.Q);
IF rtOK.Q AND q_xOverrideOpen THEN
    q_xOverrideOpen :=FALSE;
    //if (i_xOpnLS) AND (i_xOverrideMode) THEN i_xOPN_SW := TRUE; END_IF //for seamless transition
    //Log
    fbLogger(sMsg:='Override expired', eSevr:=TcEventSeverity.Warning);
END_IF
(*OPN OK evaluation bit *)
xOPN_OK := (i_xVAC_FAULT_OK) AND (NOT i_xTrigger OR (q_xVetoValveClosed AND NOT q_xVetoValveOpenDO));

(*Soft IO Mapping*)
IO();

(*Logger*)
ACT_Logger();

ACTION ACT_Logger:
//ILK logger
IF i_xTrigger AND ePrevState = OPEN THEN
         fbLogger(sMsg:='Fast valve triggered to close', eSevr:=TcEventSeverity.Critical);
END_IF

//STATE Logger
IF ePrevState <> iq_stValve.eState THEN
      CASE iq_stValve.eState OF
        INVALID:
            fbLogger(sMsg:='Valve invalid position.', eSevr:=TcEventSeverity.Critical);
          MOVING:
            fbLogger(sMsg:='Valve moving', eSevr:=TcEventSeverity.Warning);
        OPEN:
            fbLogger(sMsg:='Valve Open.', eSevr:=TcEventSeverity.Info);
        CLOSED:
            fbLogger(sMsg:='Valve closed.', eSevr:=TcEventSeverity.Info);
      END_CASE
      ePrevState := iq_stValve.eState;
  END_IF

//Log valve timeouts
tErrorPresent(CLK:=iq_stValve.bErrorPresent);
IF tErrorPresent.Q THEN fbLogger(sMsg:=iq_stValve.sErrorMessage, eSevr:=TcEventSeverity.Warning); END_IF

//Log valve open
tAction(CLK:= iq_stValve.q_xOPN_DO);
IF tAction.Q THEN fbLogger(sMsg:='Valve commanded open', eSevr:=TcEventSeverity.Info); END_IF

//Log override mode enabled
tOverrideActivated(CLK:= (tonOvrd.Q AND q_xOverrideMode));
IF tOverrideActivated.Q THEN fbLogger(sMsg:='Valve override mode activated', eSevr:=TcEventSeverity.Warning); END_IF

//Log when the trigger is vetoed
rtTriggerVetoed(CLK:= (i_xTrigger AND (NOT q_xVetoValveOpenDO AND q_xVetoValveClosed)));
IF rtTriggerVetoed.Q THEN fbLogger(sMsg:='Valve triggered while veto device is in', eSevr:=TcEventSeverity.Warning); END_IF

rtTriggered(CLK:= (i_xTrigger AND ( q_xVetoValveOpenDO AND NOT q_xVetoValveClosed)));
IF rtTriggered.Q THEN fbLogger(sMsg:='Fast valve triggered!', eSevr:=TcEventSeverity.Critical); END_IF
END_ACTION

ACTION IO:
(*inputs*)
iq_stValve.i_xTrigger := i_xTrigger;
iq_stValve.i_xOpnLS := 	i_xVFS_Open;
iq_stValve.i_xClsLS:=	i_xVFS_Closed;
iq_stValve.eVGC_State := i_eVFS_State;
iq_stValve.i_xVAC_FAULT_OK:= i_xVAC_FAULT_OK;
(*output*)
q_xOPN_SW := iq_stValve.pv_xOPN_SW;
q_xCLS_SW:= iq_stValve.xCLS_SW;
q_xVAC_FAULT_Reset :=  iq_stValve.pv_xAlmRst;
q_xOverrideMode :=iq_stValve.xOverrideMode;
q_xOverrideOpen := iq_stValve.pv_xOvrdOpn ;
iq_stValve.sGFS := CONCAT(CONCAT(CONCAT(IG1.sPath,','),CONCAT(IG2.sPath,',')),IG3.sPath);

(*Veto*)
(*VETO Devices*)
q_xVetoValveOpenDO := Veto_Valve.q_xOPN_DO;
q_xVetoValveClosed := Veto_Valve.i_xClsLS;

